KUKA KRL program: MyProgram_062().src

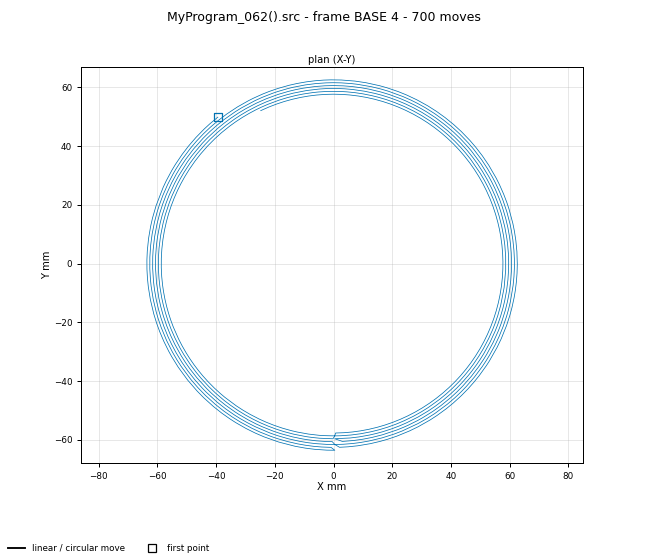
[picture p0: tool path of MyProgram_062().src in frame BASE 4, 700 of 700 moves have a stored position in this frame; points joined in program order, loops and branches not executed]
&ACCESS RVP
&REL 1
&PARAM TEMPLATE = C:\KRC\Roboter\Template\vorgabe
&PARAM EDITMASK = *
DEF MyProgram_062()
; ---- Setting reference (Base) ----
$BASE = BASE_DATA[4]

; --------------------------
; ---- Setting tool (TCP) ----
$TOOL = TOOL_DATA[3]
; --------------------------

$VEL.CP = VEL_APROX_PRINT
Startdeposition()
$VEL.CP = VEL_PRINT
LIN {X -39.4087,Y 49.8917,Z 72,A 123.1029,B 24.8681,C -2.6505,E1 24.8985,E2 -39.1381} C_DIS
LIN {X -42.1841,Y 47.5689,Z 72,A 125.8881,B 24.8698,C -2.6337,E1 24.8927,E2 -41.8942} C_DIS
LIN {X -44.0443,Y 45.8513,Z 72,A 128.1731,B 24.8703,C -2.6285,E1 24.888,E2 -44.1761} C_DIS
LIN {X -46.8498,Y 42.9805,Z 72,A 132.3088,B 24.8701,C -2.63,E1 24.88,E2 -48.3334} C_DIS
LIN {X -49.4029,Y 40.0198,Z 72,A 135.1224,B 24.8724,C -2.6071,E1 24.8751,E2 -51.1051} C_DIS
LIN {X -51.5627,Y 37.1965,Z 72,A 138.8579,B 24.8722,C -2.609,E1 24.8688,E2 -54.8631} C_DIS
LIN {X -53.8773,Y 33.7561,Z 72,A 142.4511,B 24.8735,C -2.5959,E1 24.8633,E2 -58.443} C_DIS
LIN {X -55.0548,Y 31.7997,Z 72,A 145.6129,B 24.8719,C -2.6117,E1 24.8589,E2 -61.6591} C_DIS
LIN {X -56.9529,Y 28.2593,Z 72,A 147.7032,B 24.8759,C -2.5714,E1 24.8563,E2 -63.6644} C_DIS
LIN {X -58.0502,Y 25.9311,Z 72,A 150.8815,B 24.8749,C -2.5811,E1 24.8526,E2 -66.8831} C_DIS
LIN {X -60.4404,Y 19.7284,Z 72,A 157.1125,B 24.8762,C -2.5675,E1 24.8466,E2 -73.1169} C_DIS
LIN {X -61.6489,Y 15.546,Z 72,A 160.584,B 24.8783,C -2.5466,E1 24.8441,E2 -76.5586} C_DIS
LIN {X -62.288,Y 12.7452,Z 72,A 163.2576,B 24.8789,C -2.5401,E1 24.8426,E2 -79.2325} C_DIS
LIN {X -62.9957,Y 8.5937,Z 72,A 167.1763,B 24.8798,C -2.5305,E1 24.8409,E2 -83.1516} C_DIS
LIN {X -63.432,Y 4.3135,Z 72,A 170.8648,B 24.8813,C -2.5146,E1 24.84,E2 -86.8243} C_DIS
LIN {X -63.5665,Y 1.2399,Z 72,A 173.7515,B 24.8819,C -2.508,E1 24.8398,E2 -89.7126} C_DIS
LIN {X -63.5492,Y -1.9301,Z 72,A 176.4044,B 24.8831,C -2.4951,E1 24.8399,E2 -92.3506} C_DIS
LIN {X -63.3815,Y -5.0015,Z 72,A 179.323,B 24.8837,C -2.4892,E1 24.8405,E2 -95.2727} C_DIS
LIN {X -63.0712,Y -8.0176,Z 72,A -178.3475,B 24.8852,C -2.473,E1 24.8412,E2 -97.5774} C_DIS
LIN {X -62.3757,Y -12.3121,Z 72,A -173.4784,B 24.8846,C -2.4792,E1 24.8435,E2 -102.4902} C_DIS
LIN {X -61.1949,Y -17.2459,Z 72,A -169.5379,B 24.887,C -2.4532,E1 24.8462,E2 -106.3916} C_DIS
LIN {X -60.2158,Y -20.4018,Z 72,A -166.3226,B 24.8874,C -2.4491,E1 24.849,E2 -109.6154} C_DIS
LIN {X -59.1943,Y -23.1991,Z 72,A -163.5449,B 24.888,C -2.4432,E1 24.8518,E2 -112.3946} C_DIS
LIN {X -57.8193,Y -26.4415,Z 72,A -160.1766,B 24.8884,C -2.4381,E1 24.8556,E2 -115.7694} C_DIS
LIN {X -56.1547,Y -29.8148,Z 72,A -157.088,B 24.8898,C -2.423,E1 24.8595,E2 -118.8383} C_DIS
LIN {X -55.0992,Y -31.7223,Z 72,A -154.4354,B 24.889,C -2.4315,E1 24.8633,E2 -121.5251} C_DIS
LIN {X -52.8977,Y -35.2725,Z 72,A -150.6395,B 24.8899,C -2.4226,E1 24.8691,E2 -125.3188} C_DIS
LIN {X -49.6828,Y -39.6726,Z 72,A -146.3621,B 24.8921,C -2.3981,E1 24.8762,E2 -129.5581} C_DIS
LIN {X -46.4542,Y -43.4082,Z 72,A -142.251,B 24.8936,C -2.3813,E1 24.8838,E2 -133.6478} C_DIS
LIN {X -44.2089,Y -45.6927,Z 72,A -138.8187,B 24.8931,C -2.3865,E1 24.8906,E2 -137.1067} C_DIS
LIN {X -40.9164,Y -48.6639,Z 72,A -134.084,B 24.8924,C -2.3942,E1 24.9007,E2 -141.8784} C_DIS
LIN {X -38.0706,Y -50.9204,Z 72,A -132.3527,B 24.8958,C -2.3564,E1 24.9044,E2 -143.5259} C_DIS
LIN {X -35.4553,Y -52.775,Z 72,A -129.2005,B 24.8958,C -2.3571,E1 24.9116,E2 -146.6906} C_DIS
LIN {X -33.3423,Y -54.135,Z 72,A -126.1545,B 24.8946,C -2.3702,E1 24.9189,E2 -149.7773} C_DIS
LIN {X -29.7959,Y -56.1647,Z 72,A -122.7593,B 24.8956,C -2.3592,E1 24.9271,E2 -153.156} C_DIS
LIN {X -26.6688,Y -57.7141,Z 72,A -119.8023,B 24.8962,C -2.3515,E1 24.9346,E2 -156.1024} C_DIS
LIN {X -23.6355,Y -59.0214,Z 72,A -116.2682,B 24.8954,C -2.3606,E1 24.9438,E2 -159.6661} C_DIS
LIN {X -18.6731,Y -60.7748,Z 72,A -111.3431,B 24.8954,C -2.3609,E1 24.9568,E2 -164.6009} C_DIS
LIN {X -13.1378,Y -62.2066,Z 72,A -106.4459,B 24.8961,C -2.3526,E1 24.9701,E2 -169.4849} C_DIS
LIN {X -9.5784,Y -62.853,Z 72,A -103.68,B 24.8972,C -2.3406,E1 24.9777,E2 -172.2249} C_DIS
LIN {X -6.4154,Y -63.2537,Z 72,A -100.3205,B 24.8963,C -2.3511,E1 24.9871,E2 -175.6117} C_DIS
LIN {X -2.2636,Y -63.5382,Z 72,A -97.0525,B 24.8972,C -2.3404,E1 24.9961,E2 -178.855} C_DIS
LIN {X 0.4542,Y -63.5727,Z 72,A -95.6125,B 24.8992,C -2.3181,E1 25,E2 -180.2423} C_DIS
Enddeposition()
LIN {X 0.4542,Y -63.5727,Z 72,A -95.6125,B 24.8992,C -2.3181,E1 25,E2 -180.2423} C_DIS
Startdeposition()
$VEL.CP = VEL_PRINT
LIN {X -0.8607,Y -62.5943,Z 72,A -97.3315,B 24.8987,C -2.3237,E1 24.9952,E2 -178.5364} C_DIS
LIN {X -4.0751,Y -62.4673,Z 72,A -99.6734,B 24.8976,C -2.3366,E1 24.9888,E2 -176.2246} C_DIS
LIN {X -6.8501,Y -62.2243,Z 72,A -102.6308,B 24.8983,C -2.328,E1 24.9805,E2 -173.2451} C_DIS
LIN {X -9.5335,Y -61.8698,Z 72,A -104.7295,B 24.8975,C -2.3367,E1 24.9747,E2 -171.1653} C_DIS
LIN {X -12.3094,Y -61.3778,Z 72,A -107.5509,B 24.8979,C -2.3325,E1 24.967,E2 -168.3309} C_DIS
LIN {X -15.6367,Y -60.6156,Z 72,A -111.5838,B 24.8994,C -2.3151,E1 24.9559,E2 -164.251} C_DIS
LIN {X -19.0487,Y -59.6309,Z 72,A -113.7979,B 24.8973,C -2.339,E1 24.9502,E2 -162.0898} C_DIS
LIN {X -21.296,Y -58.8665,Z 72,A -116.4905,B 24.8981,C -2.33,E1 24.943,E2 -159.3706} C_DIS
LIN {X -25.0912,Y -57.3515,Z 72,A -119.7302,B 24.8969,C -2.3441,E1 24.9347,E2 -156.1571} C_DIS
LIN {X -27.7207,Y -56.1277,Z 72,A -122.7428,B 24.8973,C -2.3399,E1 24.9271,E2 -153.1266} C_DIS
LIN {X -31.5587,Y -54.0624,Z 72,A -126.63,B 24.8966,C -2.3473,E1 24.9176,E2 -149.2459} C_DIS
LIN {X -34.5626,Y -52.1938,Z 72,A -130.121,B 24.8966,C -2.3471,E1 24.9094,E2 -145.7432} C_DIS
LIN {X -37.3656,Y -50.2258,Z 72,A -132.5987,B 24.895,C -2.3655,E1 24.9039,E2 -143.3005} C_DIS
LIN {X -40.2209,Y -47.97,Z 72,A -135.7357,B 24.8941,C -2.3753,E1 24.897,E2 -140.1753} C_DIS
LIN {X -43.5614,Y -44.9577,Z 72,A -140.7015,B 24.8949,C -2.3667,E1 24.8867,E2 -135.1691} C_DIS
LIN {X -46.1783,Y -42.265,Z 72,A -144.3865,B 24.8947,C -2.3694,E1 24.8797,E2 -131.4742} C_DIS
LIN {X -48.6608,Y -39.3813,Z 72,A -147.8735,B 24.8939,C -2.3773,E1 24.8735,E2 -127.99} C_DIS
LIN {X -51.8571,Y -35.0657,Z 72,A -152.0596,B 24.8916,C -2.4032,E1 24.8667,E2 -123.8453} C_DIS
LIN {X -53.29,Y -32.8469,Z 72,A -155.0033,B 24.892,C -2.3994,E1 24.8623,E2 -120.8775} C_DIS
LIN {X -54.8561,Y -30.1609,Z 72,A -157.6334,B 24.8909,C -2.4109,E1 24.8587,E2 -118.2612} C_DIS
LIN {X -56.8657,Y -26.173,Z 72,A -162.0699,B 24.8905,C -2.4157,E1 24.8533,E2 -113.812} C_DIS
LIN {X -58.7065,Y -21.7327,Z 72,A -166.1333,B 24.8888,C -2.4345,E1 24.8492,E2 -109.7708} C_DIS
LIN {X -59.7438,Y -18.6938,Z 72,A -168.837,B 24.8876,C -2.4475,E1 24.8468,E2 -107.0827} C_DIS
LIN {X -60.4062,Y -16.4273,Z 72,A -171.656,B 24.8881,C -2.4418,E1 24.8447,E2 -104.2338} C_DIS
LIN {X -61.4194,Y -12.1032,Z 72,A -176.6445,B 24.8885,C -2.4375,E1 24.8418,E2 -99.2056} C_DIS
LIN {X -62.1183,Y -7.7548,Z 72,A -179.0923,B 24.8847,C -2.4787,E1 24.8409,E2 -96.8416} C_DIS
LIN {X -62.3619,Y -5.4582,Z 72,A 178.1174,B 24.8852,C -2.4729,E1 24.8402,E2 -94.0208} C_DIS
LIN {X -62.5753,Y -1.7646,Z 72,A 174.8946,B 24.884,C -2.4865,E1 24.8398,E2 -90.8112} C_DIS
LIN {X -62.5603,Y 2.2343,Z 72,A 171.399,B 24.8826,C -2.5011,E1 24.84,E2 -87.3293} C_DIS
LIN {X -62.2886,Y 6.236,Z 72,A 167.1517,B 24.8825,C -2.5023,E1 24.8409,E2 -83.0593} C_DIS
LIN {X -61.7859,Y 10.066,Z 72,A 163.8912,B 24.8809,C -2.5184,E1 24.8423,E2 -79.8179} C_DIS
LIN {X -60.9672,Y 14.2046,Z 72,A 160.1823,B 24.8795,C -2.5332,E1 24.8444,E2 -76.1227} C_DIS
LIN {X -60.1472,Y 17.3504,Z 72,A 156.9368,B 24.8791,C -2.5375,E1 24.8468,E2 -72.8686} C_DIS
LIN {X -59.3158,Y 20.0098,Z 72,A 153.7977,B 24.8794,C -2.5347,E1 24.8497,E2 -69.7047} C_DIS
LIN {X -58.1418,Y 23.2013,Z 72,A 151.924,B 24.8763,C -2.5667,E1 24.8515,E2 -67.897} C_DIS
LIN {X -56.5004,Y 26.9533,Z 72,A 148.0079,B 24.8756,C -2.5747,E1 24.8559,E2 -63.9784} C_DIS
LIN {X -54.6874,Y 30.4639,Z 72,A 144.1834,B 24.8749,C -2.5812,E1 24.8609,E2 -60.1493} C_DIS
LIN {X -53.7182,Y 32.1435,Z 72,A 141.2134,B 24.8766,C -2.5643,E1 24.8653,E2 -57.1235} C_DIS
LIN {X -51.5773,Y 35.4769,Z 72,A 138.7753,B 24.8735,C -2.596,E1 24.869,E2 -54.7492} C_DIS
LIN {X -48.7578,Y 39.2617,Z 72,A 134.4087,B 24.8724,C -2.6065,E1 24.8763,E2 -50.3867} C_DIS
LIN {X -46.6518,Y 41.7416,Z 72,A 131.2568,B 24.872,C -2.6107,E1 24.8821,E2 -47.2307} C_DIS
LIN {X -44.2997,Y 44.2313,Z 72,A 128.0719,B 24.8714,C -2.6173,E1 24.8883,E2 -44.0477} C_DIS
LIN {X -41.8688,Y 46.5378,Z 72,A 124.9597,B 24.8708,C -2.6235,E1 24.8947,E2 -40.9376} C_DIS
LIN {X -39.2255,Y 48.7871,Z 72,A 120.9549,B 24.8716,C -2.6146,E1 24.9034,E2 -36.8964} C_DIS
LIN {X -36.3682,Y 50.952,Z 72,A 118.6861,B 24.8691,C -2.6406,E1 24.9084,E2 -34.6817} C_DIS
LIN {X -32.678,Y 53.3942,Z 72,A 114.9959,B 24.8676,C -2.6552,E1 24.917,E2 -31.0146} C_DIS
LIN {X -28.963,Y 55.4965,Z 72,A 110.8588,B 24.8674,C -2.6574,E1 24.9271,E2 -26.8705} C_DIS
LIN {X -27.3313,Y 56.3189,Z 72,A 108.0414,B 24.8694,C -2.6374,E1 24.9343,E2 -23.9983} C_DIS
LIN {X -24.1645,Y 57.7483,Z 72,A 106.0643,B 24.8666,C -2.6658,E1 24.9392,E2 -22.0842} C_DIS
LIN {X -21.7428,Y 58.7028,Z 72,A 102.8612,B 24.8679,C -2.6525,E1 24.9477,E2 -18.8426} C_DIS
LIN {X -18.8913,Y 59.6813,Z 72,A 100.1456,B 24.8675,C -2.6565,E1 24.9549,E2 -16.1318} C_DIS
LIN {X -15.152,Y 60.7387,Z 72,A 97.1477,B 24.866,C -2.6714,E1 24.9629,E2 -13.1648} C_DIS
LIN {X -12.5227,Y 61.3346,Z 72,A 94.1782,B 24.8668,C -2.6632,E1 24.9711,E2 -10.1722} C_DIS
LIN {X -9.2487,Y 61.9136,Z 72,A 91.6862,B 24.8655,C -2.6767,E1 24.9778,E2 -7.7101} C_DIS
LIN {X -6.2608,Y 62.2862,Z 72,A 88.4602,B 24.8663,C -2.6685,E1 24.9869,E2 -4.4623} C_DIS
LIN {X -3.3298,Y 62.5115,Z 72,A 86.2742,B 24.8651,C -2.6801,E1 24.9929,E2 -2.3033} C_DIS
LIN {X -0.8723,Y 62.5942,Z 72,A 83.5094,B 24.8661,C -2.6698,E1 25.0007,E2 0.4862} C_DIS
LIN {X 2.6652,Y 62.543,Z 72,A 79.8513,B 24.867,C -2.6613,E1 25.0109,E2 4.1638} C_DIS
LIN {X 7.2533,Y 62.1784,Z 72,A 76.2896,B 24.8657,C -2.6747,E1 25.0207,E2 7.6913} C_DIS
LIN {X 11.0314,Y 61.6203,Z 72,A 72.8045,B 24.8657,C -2.6738,E1 25.0303,E2 11.1751} C_DIS
LIN {X 15.7256,Y 60.5923,Z 72,A 68.4256,B 24.8659,C -2.672,E1 25.0422,E2 15.5523} C_DIS
LIN {X 18.2437,Y 59.8831,Z 72,A 65.6427,B 24.867,C -2.6617,E1 25.0497,E2 18.3548} C_DIS
LIN {X 22.0662,Y 58.582,Z 72,A 62.4765,B 24.8661,C -2.6703,E1 25.058,E2 21.4942} C_DIS
LIN {X 24.8618,Y 57.4515,Z 72,A 59.4177,B 24.8671,C -2.6607,E1 25.0659,E2 24.5686} C_DIS
LIN {X 28.3993,Y 55.7871,Z 72,A 55.7414,B 24.8677,C -2.6541,E1 25.0751,E2 28.2507} C_DIS
LIN {X 32.0976,Y 53.7455,Z 72,A 51.4504,B 24.8692,C -2.639,E1 25.0856,E2 32.5645} C_DIS
LIN {X 35.0671,Y 51.8561,Z 72,A 48.0357,B 24.8702,C -2.6295,E1 25.0935,E2 35.9904} C_DIS
LIN {X 38.0295,Y 49.7248,Z 72,A 45.0496,B 24.87,C -2.6317,E1 25.1001,E2 38.9602} C_DIS
LIN {X 40.9337,Y 47.3633,Z 72,A 41.7935,B 24.8702,C -2.6292,E1 25.107,E2 42.2097} C_DIS
LIN {X 43.548,Y 44.9706,Z 72,A 39.1123,B 24.8695,C -2.6358,E1 25.1124,E2 44.8642} C_DIS
LIN {X 46.4331,Y 41.9858,Z 72,A 34.8017,B 24.8716,C -2.6155,E1 25.1207,E2 49.204} C_DIS
LIN {X 48.4319,Y 39.6632,Z 72,A 31.482,B 24.8734,C -2.5969,E1 25.1266,E2 52.5526} C_DIS
LIN {X 50.6741,Y 36.7555,Z 72,A 29.5115,B 24.8709,C -2.6219,E1 25.1298,E2 54.4543} C_DIS
LIN {X 52.8826,Y 33.5001,Z 72,A 25.7875,B 24.8721,C -2.6099,E1 25.1356,E2 58.1883} C_DIS
LIN {X 55.4247,Y 29.1005,Z 72,A 21.114,B 24.8734,C -2.597,E1 25.1421,E2 62.868} C_DIS
LIN {X 56.547,Y 26.8553,Z 72,A 18.3488,B 24.8751,C -2.5793,E1 25.1455,E2 65.6603} C_DIS
LIN {X 57.9844,Y 23.5916,Z 72,A 15.3849,B 24.8753,C -2.5774,E1 25.1487,E2 68.6125} C_DIS
LIN {X 59.029,Y 20.8404,Z 72,A 12.6504,B 24.8761,C -2.5686,E1 25.1513,E2 71.3525} C_DIS
LIN {X 59.7725,Y 18.6014,Z 72,A 9.9855,B 24.8779,C -2.5498,E1 25.1536,E2 74.0466} C_DIS
LIN {X 61.0954,Y 13.6431,Z 72,A 5.9822,B 24.8777,C -2.5527,E1 25.1563,E2 78.0199} C_DIS
LIN {X 61.6136,Y 11.0689,Z 72,A 3.7892,B 24.8779,C -2.5506,E1 25.1574,E2 80.2051} C_DIS
LIN {X 62.0954,Y 7.9258,Z 72,A 0.4107,B 24.8798,C -2.53,E1 25.1588,E2 83.6126} C_DIS
LIN {X 62.4671,Y 4.0761,Z 72,A -3.3104,B 24.8813,C -2.5144,E1 25.1596,E2 87.3484} C_DIS
LIN {X 62.6,Y -0.1917,Z 72,A -6.6747,B 24.8813,C -2.5155,E1 25.1598,E2 90.69} C_DIS
LIN {X 62.5161,Y -3.2468,Z 72,A -9.7931,B 24.8828,C -2.4987,E1 25.1594,E2 93.8296} C_DIS
LIN {X 62.2941,Y -6.1801,Z 72,A -12.0861,B 24.8827,C -2.5001,E1 25.1589,E2 96.1057} C_DIS
LIN {X 61.9148,Y -9.2354,Z 72,A -15.0389,B 24.8838,C -2.4878,E1 25.1578,E2 99.0701} C_DIS
LIN {X 61.5276,Y -11.5374,Z 72,A -17.3677,B 24.8849,C -2.4763,E1 25.1566,E2 101.4125} C_DIS
LIN {X 60.7674,Y -15.0373,Z 72,A -20.3845,B 24.8853,C -2.4725,E1 25.1547,E2 104.4206} C_DIS
LIN {X 60.0254,Y -17.7675,Z 72,A -23.0144,B 24.8861,C -2.4635,E1 25.1527,E2 107.0568} C_DIS
LIN {X 58.9462,Y -21.0734,Z 72,A -26.5582,B 24.8878,C -2.4448,E1 25.1495,E2 110.6248} C_DIS
LIN {X 57.1353,Y -25.5792,Z 72,A -30.7757,B 24.8885,C -2.4371,E1 25.1449,E2 114.8374} C_DIS
LIN {X 55.7289,Y -28.5139,Z 72,A -34.274,B 24.8905,C -2.4156,E1 25.1405,E2 118.3678} C_DIS
LIN {X 53.0584,Y -33.22,Z 72,A -38.2032,B 24.8895,C -2.4267,E1 25.135,E2 122.2506} C_DIS
LIN {X 52.1163,Y -34.6802,Z 72,A -40.0053,B 24.8904,C -2.4171,E1 25.1322,E2 124.0665} C_DIS
LIN {X 49.6583,Y -38.116,Z 72,A -43.5616,B 24.8906,C -2.4143,E1 25.1264,E2 127.6122} C_DIS
LIN {X 47.8309,Y -40.3853,Z 72,A -46.5328,B 24.8919,C -2.4,E1 25.1211,E2 130.6036} C_DIS
LIN {X 45.7888,Y -42.6851,Z 72,A -49.5818,B 24.8931,C -2.3873,E1 25.1153,E2 133.669} C_DIS
LIN {X 43.5354,Y -44.9827,Z 72,A -52.2506,B 24.8931,C -2.3869,E1 25.11,E2 136.3275} C_DIS
LIN {X 40.7303,Y -47.5376,Z 72,A -55.8059,B 24.894,C -2.3771,E1 25.1026,E2 139.892} C_DIS
LIN {X 38.3574,Y -49.471,Z 72,A -58.6663,B 24.8946,C -2.3697,E1 25.0963,E2 142.7592} C_DIS
LIN {X 35.23,Y -51.7458,Z 72,A -62.4022,B 24.8957,C -2.3579,E1 25.0877,E2 146.5101} C_DIS
LIN {X 32.8782,Y -53.2717,Z 72,A -64.9739,B 24.8961,C -2.353,E1 25.0816,E2 149.0852} C_DIS
LIN {X 28.8443,Y -55.5589,Z 72,A -69.631,B 24.8976,C -2.3362,E1 25.0701,E2 153.7688} C_DIS
LIN {X 25.8402,Y -57.0179,Z 72,A -71.6799,B 24.8959,C -2.3548,E1 25.0651,E2 155.7682} C_DIS
LIN {X 21.5781,Y -58.7636,Z 72,A -75.5966,B 24.8959,C -2.3559,E1 25.055,E2 159.6735} C_DIS
LIN {X 18.3344,Y -59.855,Z 72,A -79.2874,B 24.8973,C -2.3393,E1 25.0451,E2 163.3968} C_DIS
LIN {X 15.8373,Y -60.5637,Z 72,A -81.3397,B 24.8969,C -2.3442,E1 25.0396,E2 165.4342} C_DIS
LIN {X 12.4936,Y -61.3406,Z 72,A -84.1303,B 24.8964,C -2.3493,E1 25.032,E2 168.2088} C_DIS
LIN {X 8.3178,Y -62.0451,Z 72,A -88.061,B 24.8968,C -2.3451,E1 25.0212,E2 172.1454} C_DIS
LIN {X 4.9941,Y -62.4004,Z 72,A -91.6246,B 24.8979,C -2.3321,E1 25.0112,E2 175.7375} C_DIS
LIN {X 2.0567,Y -62.5663,Z 72,A -94.284,B 24.8979,C -2.3319,E1 25.0038,E2 178.3967} C_DIS
LIN {X 2.0567,Y -62.5663,Z 72,A -94.284,B 24.8979,C -2.3319,E1 25.0038,E2 178.3967} C_DIS
Enddeposition()
LIN {X 0.4424,Y -61.6194,Z 72,A -94.8099,B 24.8946,C -2.3694,E1 25.0026,E2 178.8334} C_DIS
Startdeposition()
$VEL.CP = VEL_PRINT
LIN {X 3.293,Y -61.5335,Z 72,A -91.6913,B 24.8936,C -2.3808,E1 25.0113,E2 175.6887} C_DIS
LIN {X 6.3281,Y -61.2955,Z 72,A -89.1713,B 24.8941,C -2.3753,E1 25.0183,E2 173.1833} C_DIS
LIN {X 8.8597,Y -60.9812,Z 72,A -85.9133,B 24.8922,C -2.397,E1 25.0274,E2 169.8766} C_DIS
LIN {X 12.0469,Y -60.4326,Z 72,A -83.4386,B 24.8931,C -2.3872,E1 25.0342,E2 167.4279} C_DIS
LIN {X 16.4999,Y -59.3717,Z 72,A -79.4267,B 24.8931,C -2.3859,E1 25.045,E2 163.4253} C_DIS
LIN {X 20.7143,Y -58.0354,Z 72,A -75.3956,B 24.8929,C -2.389,E1 25.0557,E2 159.3945} C_DIS
LIN {X 23.374,Y -57.016,Z 72,A -72.5319,B 24.8921,C -2.3977,E1 25.0631,E2 156.5167} C_DIS
LIN {X 28.7742,Y -54.4908,Z 72,A -67.1581,B 24.8917,C -2.4024,E1 25.0766,E2 151.1458} C_DIS
LIN {X 31.8208,Y -52.7698,Z 72,A -64.1285,B 24.8917,C -2.4029,E1 25.0839,E2 148.1241} C_DIS
LIN {X 34.5048,Y -51.0551,Z 72,A -60.468,B 24.8896,C -2.4254,E1 25.0926,E2 144.4227} C_DIS
LIN {X 38.7763,Y -47.8915,Z 72,A -56.1143,B 24.89,C -2.4215,E1 25.1021,E2 140.094} C_DIS
LIN {X 41.3572,Y -45.6824,Z 72,A -52.9013,B 24.8892,C -2.4299,E1 25.1089,E2 136.8737} C_DIS
LIN {X 43.5322,Y -43.6148,Z 72,A -50.4166,B 24.8892,C -2.4291,E1 25.1139,E2 134.4013} C_DIS
LIN {X 45.2616,Y -41.8163,Z 72,A -47.9192,B 24.8883,C -2.4391,E1 25.1187,E2 131.8911} C_DIS
LIN {X 48.0068,Y -38.6341,Z 72,A -44.0033,B 24.8874,C -2.4493,E1 25.1257,E2 127.969} C_DIS
LIN {X 50.6737,Y -35.0628,Z 72,A -39.8495,B 24.8864,C -2.4607,E1 25.1326,E2 123.8084} C_DIS
LIN {X 52.0159,Y -33.0396,Z 72,A -37.923,B 24.8865,C -2.4588,E1 25.1355,E2 121.896} C_DIS
LIN {X 53.2021,Y -31.0939,Z 72,A -35.2638,B 24.8847,C -2.4782,E1 25.1393,E2 119.2047} C_DIS
LIN {X 55.0274,Y -27.7343,Z 72,A -32.2869,B 24.8851,C -2.4741,E1 25.1432,E2 116.2529} C_DIS
LIN {X 56.3578,Y -24.9191,Z 72,A -28.8028,B 24.8829,C -2.4974,E1 25.1473,E2 112.7329} C_DIS
LIN {X 57.7739,Y -21.4335,Z 72,A -25.1084,B 24.8815,C -2.5129,E1 25.151,E2 109.0223} C_DIS
LIN {X 58.9461,Y -17.9613,Z 72,A -22.3487,B 24.882,C -2.5071,E1 25.1533,E2 106.2919} C_DIS
LIN {X 59.5578,Y -15.8146,Z 72,A -20.3456,B 24.8816,C -2.5118,E1 25.1548,E2 104.2893} C_DIS
LIN {X 60.2468,Y -12.9414,Z 72,A -16.9379,B 24.8792,C -2.5369,E1 25.1569,E2 100.8418} C_DIS
LIN {X 61.1682,Y -7.4614,Z 72,A -12.2619,B 24.8788,C -2.5409,E1 25.1588,E2 96.1841} C_DIS
LIN {X 61.4634,Y -4.418,Z 72,A -9.4833,B 24.8781,C -2.5483,E1 25.1595,E2 93.4045} C_DIS
LIN {X 61.6017,Y -1.5586,Z 72,A -6.4637,B 24.8764,C -2.5657,E1 25.1598,E2 90.3617} C_DIS
LIN {X 61.5989,Y 1.6666,Z 72,A -4.1806,B 24.8772,C -2.5573,E1 25.1597,E2 88.112} C_DIS
LIN {X 61.4573,Y 4.4916,Z 72,A -1.1094,B 24.8754,C -2.5765,E1 25.1592,E2 85.0136} C_DIS
LIN {X 61.0842,Y 8.119,Z 72,A 2.4249,B 24.874,C -2.5907,E1 25.158,E2 81.4668} C_DIS
LIN {X 60.553,Y 11.426,Z 72,A 5.0789,B 24.8742,C -2.5888,E1 25.1567,E2 78.8328} C_DIS
LIN {X 60.1363,Y 13.4477,Z 72,A 7.4108,B 24.8726,C -2.6049,E1 25.1553,E2 76.4764} C_DIS
LIN {X 59.0332,Y 17.6704,Z 72,A 11.1983,B 24.8721,C -2.6103,E1 25.1525,E2 72.6978} C_DIS
LIN {X 57.676,Y 21.6935,Z 72,A 15.2338,B 24.8707,C -2.6239,E1 25.1487,E2 68.6527} C_DIS
LIN {X 56.5416,Y 24.4988,Z 72,A 18.0173,B 24.87,C -2.6311,E1 25.1457,E2 65.8674} C_DIS
LIN {X 55.1024,Y 27.5861,Z 72,A 20.8147,B 24.87,C -2.6308,E1 25.1424,E2 63.0859} C_DIS
LIN {X 54.1468,Y 29.4162,Z 72,A 23.7492,B 24.8671,C -2.6608,E1 25.1384,E2 60.0957} C_DIS
LIN {X 52.4711,Y 32.312,Z 72,A 25.6755,B 24.8691,C -2.64,E1 25.1357,E2 58.2286} C_DIS
LIN {X 50.4861,Y 35.3319,Z 72,A 29.2782,B 24.8677,C -2.6543,E1 25.1301,E2 54.6099} C_DIS
LIN {X 47.7248,Y 38.982,Z 72,A 33.303,B 24.8673,C -2.6588,E1 25.1232,E2 50.5935} C_DIS
LIN {X 45.9258,Y 41.0855,Z 72,A 36.3387,B 24.8656,C -2.6756,E1 25.1176,E2 47.5316} C_DIS
LIN {X 42.9113,Y 44.2251,Z 72,A 39.7296,B 24.8663,C -2.6686,E1 25.111,E2 44.1718} C_DIS
LIN {X 40.2688,Y 46.6447,Z 72,A 43.5083,B 24.8646,C -2.6857,E1 25.1031,E2 40.3679} C_DIS
LIN {X 37.3257,Y 49.0314,Z 72,A 47.7007,B 24.8623,C -2.7077,E1 25.0938,E2 36.1387} C_DIS
LIN {X 34.4428,Y 51.0971,Z 72,A 50.2908,B 24.8634,C -2.6965,E1 25.088,E2 33.584} C_DIS
LIN {X 31.1518,Y 53.1679,Z 72,A 53.8399,B 24.8631,C -2.7003,E1 25.0795,E2 30.037} C_DIS
LIN {X 28.6727,Y 54.5439,Z 72,A 56.4622,B 24.8627,C -2.7035,E1 25.0731,E2 27.4147} C_DIS
LIN {X 26.3301,Y 55.7131,Z 72,A 59.3059,B 24.8615,C -2.7158,E1 25.0659,E2 24.5493} C_DIS
LIN {X 23.6707,Y 56.8941,Z 72,A 61.9784,B 24.8613,C -2.7178,E1 25.059,E2 21.8782} C_DIS
LIN {X 18.6415,Y 58.734,Z 72,A 66.6013,B 24.8617,C -2.7141,E1 25.0469,E2 17.2736} C_DIS
LIN {X 16.1745,Y 59.4609,Z 72,A 69.8633,B 24.8595,C -2.7351,E1 25.038,E2 13.967} C_DIS
LIN {X 12.9038,Y 60.2554,Z 72,A 71.8664,B 24.8619,C -2.7117,E1 25.0327,E2 12.0222} C_DIS
LIN {X 8.0374,Y 61.095,Z 72,A 76.7686,B 24.8611,C -2.7198,E1 25.0191,E2 7.1054} C_DIS
LIN {X 5.9705,Y 61.3315,Z 72,A 78.9371,B 24.8605,C -2.7251,E1 25.013,E2 4.9257} C_DIS
LIN {X 2.6608,Y 61.564,Z 72,A 81.6397,B 24.8614,C -2.7169,E1 25.0056,E2 2.2438} C_DIS
LIN {X -0.0111,Y 61.6214,Z 72,A 84.4185,B 24.8608,C -2.7227,E1 24.9978,E2 -0.5487} C_DIS
LIN {X -2.5835,Y 61.5673,Z 72,A 86.3775,B 24.8618,C -2.7128,E1 24.9924,E2 -2.4844} C_DIS
LIN {X -6.015,Y 61.3271,Z 72,A 90.3145,B 24.8603,C -2.7269,E1 24.9813,E2 -6.4568} C_DIS
LIN {X -9.5739,Y 60.8734,Z 72,A 93.4785,B 24.8609,C -2.7211,E1 24.9726,E2 -9.6096} C_DIS
LIN {X -13.8436,Y 60.0462,Z 72,A 97.0824,B 24.8622,C -2.7087,E1 24.9628,E2 -13.1881} C_DIS
LIN {X -15.5319,Y 59.632,Z 72,A 98.6849,B 24.8624,C -2.7068,E1 24.9585,E2 -14.7885} C_DIS
LIN {X -19.0868,Y 58.5911,Z 72,A 102.0793,B 24.8629,C -2.702,E1 24.9494,E2 -18.1773} C_DIS
LIN {X -20.8304,Y 57.9936,Z 72,A 104.545,B 24.8616,C -2.7151,E1 24.9429,E2 -20.6791} C_DIS
LIN {X -24.2643,Y 56.6433,Z 72,A 107.5496,B 24.8629,C -2.7017,E1 24.9352,E2 -23.6586} C_DIS
LIN {X -26.8,Y 55.4885,Z 72,A 110.4436,B 24.8627,C -2.7038,E1 24.9278,E2 -26.5649} C_DIS
LIN {X -31.3577,Y 53.0462,Z 72,A 114.2983,B 24.8654,C -2.6769,E1 24.9185,E2 -30.3664} C_DIS
LIN {X -33.4403,Y 51.7589,Z 72,A 117.5929,B 24.8638,C -2.6926,E1 24.9107,E2 -33.709} C_DIS
LIN {X -37.2722,Y 49.0717,Z 72,A 121.9127,B 24.8648,C -2.6832,E1 24.9009,E2 -38.0214} C_DIS
LIN {X -39.843,Y 47.0081,Z 72,A 124.4813,B 24.8664,C -2.6669,E1 24.8955,E2 -40.5611} C_DIS
LIN {X -42.17,Y 44.9321,Z 72,A 127.7734,B 24.8664,C -2.6679,E1 24.8886,E2 -43.8687} C_DIS
LIN {X -44.4139,Y 42.7155,Z 72,A 131.1914,B 24.8661,C -2.6702,E1 24.882,E2 -47.3069} C_DIS
LIN {X -47.6724,Y 39.0462,Z 72,A 135.4264,B 24.8679,C -2.6523,E1 24.8743,E2 -51.5186} C_DIS
LIN {X -50.2791,Y 35.6265,Z 72,A 138.6832,B 24.8703,C -2.6278,E1 24.869,E2 -54.7325} C_DIS
LIN {X -51.9739,Y 33.1044,Z 72,A 142.2846,B 24.8697,C -2.6345,E1 24.8634,E2 -58.3681} C_DIS
LIN {X -53.5263,Y 30.5316,Z 72,A 144.9196,B 24.8708,C -2.6236,E1 24.8597,E2 -60.9907} C_DIS
LIN {X -55.1466,Y 27.4967,Z 72,A 148.0249,B 24.8718,C -2.6126,E1 24.8558,E2 -64.0863} C_DIS
LIN {X -56.9819,Y 23.4582,Z 72,A 151.7849,B 24.8737,C -2.5936,E1 24.8516,E2 -67.8216} C_DIS
LIN {X -58.1857,Y 20.2882,Z 72,A 155.2559,B 24.8741,C -2.5899,E1 24.8482,E2 -71.3033} C_DIS
LIN {X -59.1408,Y 17.3073,Z 72,A 158.6312,B 24.8741,C -2.5896,E1 24.8454,E2 -74.6972} C_DIS
LIN {X -60.1167,Y 13.533,Z 72,A 162.1316,B 24.8754,C -2.576,E1 24.8431,E2 -78.1856} C_DIS
LIN {X -60.9482,Y 9.0903,Z 72,A 166.5285,B 24.8764,C -2.5663,E1 24.8411,E2 -82.5855} C_DIS
LIN {X -61.4507,Y 4.5758,Z 72,A 170.3764,B 24.8783,C -2.546,E1 24.8401,E2 -86.408} C_DIS
LIN {X -61.5777,Y 2.3158,Z 72,A 172.8124,B 24.8783,C -2.5455,E1 24.8398,E2 -88.8574} C_DIS
LIN {X -61.6007,Y -1.599,Z 72,A 176.3491,B 24.8796,C -2.5321,E1 24.8399,E2 -92.3834} C_DIS
LIN {X -61.3299,Y -5.9873,Z 72,A -179.9999,B 24.8816,C -2.5112,E1 24.8407,E2 -96.0064} C_DIS
LIN {X -60.9823,Y -8.8504,Z 72,A -176.2101,B 24.8805,C -2.5235,E1 24.8421,E2 -99.8481} C_DIS
LIN {X -60.4282,Y -12.0684,Z 72,A -173.0311,B 24.8811,C -2.5169,E1 24.8439,E2 -103.0301} C_DIS
LIN {X -59.6384,Y -15.5077,Z 72,A -170.646,B 24.8836,C -2.4902,E1 24.8455,E2 -105.3655} C_DIS
LIN {X -58.8223,Y -18.3618,Z 72,A -168.2141,B 24.8849,C -2.4759,E1 24.8474,E2 -107.7773} C_DIS
LIN {X -57.7758,Y -21.4285,Z 72,A -164.593,B 24.8847,C -2.4785,E1 24.8508,E2 -111.4251} C_DIS
LIN {X -56.3649,Y -24.9032,Z 72,A -161.4957,B 24.8863,C -2.4614,E1 24.8541,E2 -114.4986} C_DIS
LIN {X -55.1867,Y -27.4157,Z 72,A -158.408,B 24.8861,C -2.4639,E1 24.8579,E2 -117.609} C_DIS
LIN {X -53.6625,Y -30.2922,Z 72,A -155.7878,B 24.8875,C -2.448,E1 24.8614,E2 -120.2052} C_DIS
LIN {X -51.706,Y -33.5227,Z 72,A -152.0795,B 24.888,C -2.4428,E1 24.8669,E2 -123.9198} C_DIS
LIN {X -49.5583,Y -36.623,Z 72,A -147.8818,B 24.8876,C -2.4476,E1 24.8738,E2 -128.1496} C_DIS
LIN {X -47.2847,Y -39.5144,Z 72,A -145.1933,B 24.8896,C -2.4255,E1 24.8785,E2 -130.7977} C_DIS
LIN {X -44.7547,Y -42.3586,Z 72,A -141.5998,B 24.8902,C -2.4188,E1 24.8852,E2 -134.391} C_DIS
LIN {X -43.3675,Y -43.7775,Z 72,A -139.5495,B 24.8902,C -2.419,E1 24.8893,E2 -136.4506} C_DIS
LIN {X -39.6704,Y -47.1545,Z 72,A -134.629,B 24.8905,C -2.4153,E1 24.8996,E2 -141.3817} C_DIS
LIN {X -36.6602,Y -49.5308,Z 72,A -131.2398,B 24.8914,C -2.4056,E1 24.9071,E2 -144.7599} C_DIS
LIN {X -33.609,Y -51.6501,Z 72,A -128.2464,B 24.8927,C -2.3908,E1 24.914,E2 -147.7281} C_DIS
LIN {X -31.8463,Y -52.7546,Z 72,A -126.0736,B 24.8926,C -2.3928,E1 24.9192,E2 -149.9124} C_DIS
LIN {X -29.2655,Y -54.2287,Z 72,A -123.0014,B 24.8923,C -2.3955,E1 24.9268,E2 -152.9999} C_DIS
LIN {X -26.6277,Y -55.5713,Z 72,A -120.2987,B 24.8927,C -2.3912,E1 24.9335,E2 -155.6994} C_DIS
LIN {X -21.7331,Y -57.6618,Z 72,A -115.6451,B 24.8937,C -2.3802,E1 24.9455,E2 -160.337} C_DIS
LIN {X -19.1426,Y -58.5729,Z 72,A -112.5287,B 24.8928,C -2.39,E1 24.9539,E2 -163.4828} C_DIS
LIN {X -15.4327,Y -59.6577,Z 72,A -109.8105,B 24.8947,C -2.3692,E1 24.961,E2 -166.1556} C_DIS
LIN {X -11.4757,Y -60.5436,Z 72,A -105.7407,B 24.8943,C -2.3739,E1 24.9722,E2 -170.2416} C_DIS
LIN {X -8.8672,Y -60.9803,Z 72,A -103.252,B 24.8943,C -2.3739,E1 24.9791,E2 -172.7324} C_DIS
LIN {X -6.1503,Y -61.3135,Z 72,A -100.5068,B 24.8939,C -2.378,E1 24.9867,E2 -175.489} C_DIS
LIN {X -2.1776,Y -61.583,Z 72,A -96.959,B 24.8942,C -2.3748,E1 24.9966,E2 -179.0302} C_DIS
LIN {X 0.4424,Y -61.6194,Z 72,A -94.8089,B 24.8947,C -2.369,E1 25.0026,E2 -181.1666} C_DIS
Enddeposition()
LIN {X 0.4424,Y -61.6194,Z 72,A -94.8089,B 24.8947,C -2.369,E1 25.0026,E2 -181.1666} C_DIS
Startdeposition()
$VEL.CP = VEL_PRINT
LIN {X -0.4328,Y -60.6414,Z 72,A -96.3852,B 24.8947,C -2.3695,E1 24.9982,E2 -179.5916} C_DIS
LIN {X -2.7331,Y -60.5813,Z 72,A -98.9926,B 24.8955,C -2.3601,E1 24.9908,E2 -176.9614} C_DIS
LIN {X -5.8894,Y -60.3562,Z 72,A -101.8982,B 24.8953,C -2.362,E1 24.9827,E2 -174.0588} C_DIS
LIN {X -9.0908,Y -59.9579,Z 72,A -104.6176,B 24.8947,C -2.3694,E1 24.9753,E2 -171.355} C_DIS
LIN {X -10.6356,Y -59.703,Z 72,A -107.2508,B 24.8967,C -2.3462,E1 24.9679,E2 -168.664} C_DIS
LIN {X -13.9347,Y -59.0203,Z 72,A -109.4776,B 24.8949,C -2.3672,E1 24.9619,E2 -166.4842} C_DIS
LIN {X -18.0565,Y -57.8924,Z 72,A -113.556,B 24.8947,C -2.3689,E1 24.951,E2 -162.4035} C_DIS
LIN {X -20.6285,Y -57.0268,Z 72,A -116.1965,B 24.8947,C -2.3695,E1 24.944,E2 -159.7592} C_DIS
LIN {X -24.3677,Y -55.532,Z 72,A -120.0469,B 24.8944,C -2.3724,E1 24.9341,E2 -155.907} C_DIS
LIN {X -26.2762,Y -54.6546,Z 72,A -122.1833,B 24.8944,C -2.3717,E1 24.9287,E2 -153.7635} C_DIS
LIN {X -28.9999,Y -53.2595,Z 72,A -124.9843,B 24.894,C -2.3772,E1 24.9218,E2 -150.9677} C_DIS
LIN {X -32.1384,Y -51.4265,Z 72,A -127.8567,B 24.8925,C -2.393,E1 24.9149,E2 -148.1243} C_DIS
LIN {X -33.5087,Y -50.5446,Z 72,A -130.5736,B 24.8944,C -2.3727,E1 24.9085,E2 -145.3501} C_DIS
LIN {X -36.7046,Y -48.2743,Z 72,A -133.427,B 24.8923,C -2.3952,E1 24.9022,E2 -142.5402} C_DIS
LIN {X -38.9375,Y -46.4918,Z 72,A -137.221,B 24.8937,C -2.3795,E1 24.8939,E2 -138.6943} C_DIS
LIN {X -41.5169,Y -44.203,Z 72,A -139.2805,B 24.8911,C -2.4084,E1 24.8898,E2 -136.6954} C_DIS
LIN {X -43.095,Y -42.666,Z 72,A -141.6989,B 24.8913,C -2.4064,E1 24.885,E2 -134.262} C_DIS
LIN {X -46.5456,Y -38.8727,Z 72,A -147.5882,B 24.8921,C -2.398,E1 24.8741,E2 -128.3261} C_DIS
LIN {X -48.8597,Y -35.9208,Z 72,A -150.1623,B 24.8897,C -2.4242,E1 24.8699,E2 -125.802} C_DIS
LIN {X -50.4287,Y -33.6833,Z 72,A -152.5404,B 24.8888,C -2.4343,E1 24.8661,E2 -123.4363} C_DIS
LIN {X -51.8872,Y -31.3894,Z 72,A -155.5178,B 24.8888,C -2.4334,E1 24.8617,E2 -120.4417} C_DIS
LIN {X -54.1033,Y -27.3928,Z 72,A -159.8534,B 24.8878,C -2.4447,E1 24.856,E2 -116.11} C_DIS
LIN {X -55.4885,Y -24.4646,Z 72,A -162.8288,B 24.8869,C -2.4548,E1 24.8526,E2 -113.1424} C_DIS
LIN {X -56.845,Y -21.1242,Z 72,A -166.4192,B 24.8863,C -2.4612,E1 24.8489,E2 -109.5472} C_DIS
LIN {X -58.0089,Y -17.68,Z 72,A -169.6731,B 24.8851,C -2.4745,E1 24.8462,E2 -106.3066} C_DIS
LIN {X -58.8306,Y -14.7153,Z 72,A -173.0985,B 24.8851,C -2.4741,E1 24.8438,E2 -102.8602} C_DIS
LIN {X -59.4918,Y -11.7621,Z 72,A -175.9769,B 24.8843,C -2.4825,E1 24.8422,E2 -99.9848} C_DIS
LIN {X -60.2856,Y -6.5758,Z 72,A 179.848,B 24.8816,C -2.5116,E1 24.8406,E2 -95.8543} C_DIS
LIN {X -60.6178,Y -1.746,Z 72,A 175.3432,B 24.8801,C -2.5271,E1 24.8398,E2 -91.3596} C_DIS
LIN {X -60.5848,Y 2.6542,Z 72,A 170.7876,B 24.8795,C -2.5333,E1 24.84,E2 -86.7912} C_DIS
LIN {X -60.2966,Y 6.4718,Z 72,A 166.7466,B 24.8791,C -2.5373,E1 24.8411,E2 -82.7356} C_DIS
LIN {X -59.954,Y 9.1161,Z 72,A 164.1807,B 24.8785,C -2.5444,E1 24.8421,E2 -80.1714} C_DIS
LIN {X -59.0666,Y 13.7369,Z 72,A 160.2118,B 24.8763,C -2.5667,E1 24.8444,E2 -76.2323} C_DIS
LIN {X -58.3667,Y 16.4588,Z 72,A 157.079,B 24.8763,C -2.5666,E1 24.8467,E2 -73.081} C_DIS
LIN {X -57.0484,Y 20.5684,Z 72,A 153.0859,B 24.875,C -2.5805,E1 24.8502,E2 -69.0985} C_DIS
LIN {X -56.0088,Y 23.251,Z 72,A 150.2692,B 24.8744,C -2.5869,E1 24.8532,E2 -66.2814} C_DIS
LIN {X -54.1509,Y 27.2991,Z 72,A 146.3305,B 24.8727,C -2.604,E1 24.8579,E2 -62.3622} C_DIS
LIN {X -52.7864,Y 29.854,Z 72,A 143.5752,B 24.872,C -2.6115,E1 24.8616,E2 -59.6103} C_DIS
LIN {X -49.763,Y 34.6584,Z 72,A 138.6903,B 24.8696,C -2.6349,E1 24.869,E2 -54.7566} C_DIS
LIN {X -48.27,Y 36.7088,Z 72,A 135.173,B 24.871,C -2.6211,E1 24.8749,E2 -51.1895} C_DIS
LIN {X -44.7539,Y 40.9227,Z 72,A 130.2797,B 24.8692,C -2.6394,E1 24.8838,E2 -46.3177} C_DIS
LIN {X -42.9306,Y 42.8324,Z 72,A 127.6835,B 24.8688,C -2.6435,E1 24.889,E2 -43.7202} C_DIS
LIN {X -39.4157,Y 46.0866,Z 72,A 123.8777,B 24.8664,C -2.6669,E1 24.8968,E2 -39.9551} C_DIS
LIN {X -37.0729,Y 47.9913,Z 72,A 120.3861,B 24.867,C -2.6611,E1 24.9044,E2 -36.4368} C_DIS
LIN {X -35.0605,Y 49.481,Z 72,A 117.5028,B 24.8675,C -2.6563,E1 24.9111,E2 -33.5319} C_DIS
LIN {X -32.3761,Y 51.2779,Z 72,A 115.2898,B 24.8654,C -2.6776,E1 24.9162,E2 -31.3626} C_DIS
LIN {X -29.8954,Y 52.7631,Z 72,A 112.0447,B 24.8659,C -2.6727,E1 24.9241,E2 -28.0962} C_DIS
LIN {X -26.2686,Y 54.6582,Z 72,A 108.2946,B 24.865,C -2.681,E1 24.9334,E2 -24.356} C_DIS
LIN {X -22.8901,Y 56.157,Z 72,A 104.3223,B 24.8654,C -2.6768,E1 24.9437,E2 -20.3646} C_DIS
LIN {X -18.8542,Y 57.6376,Z 72,A 100.0487,B 24.8654,C -2.6775,E1 24.955,E2 -16.0848} C_DIS
LIN {X -15.3634,Y 58.6647,Z 72,A 98.0524,B 24.8622,C -2.7092,E1 24.9602,E2 -14.1606} C_DIS
LIN {X -12.9788,Y 59.2377,Z 72,A 95.3048,B 24.8628,C -2.7027,E1 24.9677,E2 -11.3941} C_DIS
LIN {X -10.3855,Y 59.7472,Z 72,A 92.7515,B 24.8628,C -2.7035,E1 24.9747,E2 -8.84} C_DIS
LIN {X -6.2395,Y 60.3209,Z 72,A 88.4485,B 24.8632,C -2.6988,E1 24.9867,E2 -4.5229} C_DIS
LIN {X -2.9521,Y 60.5712,Z 72,A 86.0454,B 24.8616,C -2.7145,E1 24.9933,E2 -2.1562} C_DIS
LIN {X -0.1188,Y 60.6425,Z 72,A 82.8612,B 24.8626,C -2.7048,E1 25.0022,E2 1.0512} C_DIS
LIN {X 3.3413,Y 60.5507,Z 72,A 79.5244,B 24.8627,C -2.7036,E1 25.0115,E2 4.3898} C_DIS
LIN {X 6.2118,Y 60.324,Z 72,A 77.3279,B 24.8616,C -2.7143,E1 25.0176,E2 6.5598} C_DIS
LIN {X 9.6594,Y 59.868,Z 72,A 73.5503,B 24.8628,C -2.7031,E1 25.0281,E2 10.3605} C_DIS
LIN {X 12.0804,Y 59.4274,Z 72,A 70.6627,B 24.8641,C -2.6903,E1 25.0361,E2 13.275} C_DIS
LIN {X 16.1002,Y 58.4668,Z 72,A 67.5052,B 24.8627,C -2.7038,E1 25.0445,E2 16.3957} C_DIS
LIN {X 18.989,Y 57.5934,Z 72,A 64.2498,B 24.8638,C -2.6929,E1 25.0532,E2 19.6708} C_DIS
LIN {X 22.7628,Y 56.2088,Z 72,A 61.2862,B 24.8623,C -2.7074,E1 25.0608,E2 22.5936} C_DIS
LIN {X 24.9929,Y 55.2528,Z 72,A 58.7379,B 24.8632,C -2.6993,E1 25.0674,E2 25.1549} C_DIS
LIN {X 27.4251,Y 54.087,Z 72,A 55.9233,B 24.8641,C -2.6904,E1 25.0745,E2 27.9833} C_DIS
LIN {X 29.7761,Y 52.83,Z 72,A 53.8507,B 24.8634,C -2.6968,E1 25.0795,E2 30.0345} C_DIS
LIN {X 31.7154,Y 51.6891,Z 72,A 50.9354,B 24.8655,C -2.6762,E1 25.0866,E2 32.9896} C_DIS
LIN {X 34.7349,Y 49.7098,Z 72,A 47.6265,B 24.8658,C -2.673,E1 25.0942,E2 36.295} C_DIS
LIN {X 38.1064,Y 47.1749,Z 72,A 43.8446,B 24.8661,C -2.6704,E1 25.1025,E2 40.0689} C_DIS
LIN {X 40.9781,Y 44.703,Z 72,A 40.4563,B 24.8663,C -2.6678,E1 25.1096,E2 43.45} C_DIS
LIN {X 43.1665,Y 42.5936,Z 72,A 36.7997,B 24.8687,C -2.644,E1 25.1169,E2 47.1475} C_DIS
LIN {X 45.4182,Y 40.1846,Z 72,A 34.5253,B 24.8675,C -2.6563,E1 25.121,E2 49.3826} C_DIS
LIN {X 47.0016,Y 38.3203,Z 72,A 31.617,B 24.8694,C -2.6372,E1 25.1262,E2 52.3226} C_DIS
LIN {X 50.2947,Y 33.882,Z 72,A 26.6297,B 24.8701,C -2.6298,E1 25.1343,E2 57.3032} C_DIS
LIN {X 52.8512,Y 29.7363,Z 72,A 22.4626,B 24.8703,C -2.628,E1 25.1402,E2 61.4532} C_DIS
LIN {X 53.9467,Y 27.7007,Z 72,A 20.372,B 24.8707,C -2.6243,E1 25.1429,E2 63.5416} C_DIS
LIN {X 55.1032,Y 25.3216,Z 72,A 17.4418,B 24.8724,C -2.6072,E1 25.1464,E2 66.4963} C_DIS
LIN {X 56.5551,Y 21.8871,Z 72,A 14.1808,B 24.8728,C -2.6034,E1 25.1498,E2 69.7484} C_DIS
LIN {X 57.532,Y 19.175,Z 72,A 11.5942,B 24.8732,C -2.5987,E1 25.1522,E2 72.3316} C_DIS
LIN {X 58.7031,Y 15.2139,Z 72,A 7.4716,B 24.8749,C -2.5818,E1 25.1553,E2 76.4704} C_DIS
LIN {X 59.372,Y 12.3511,Z 72,A 4.8818,B 24.8752,C -2.5778,E1 25.1569,E2 79.0546} C_DIS
LIN {X 59.9099,Y 9.4007,Z 72,A 2.13,B 24.8759,C -2.5711,E1 25.1581,E2 81.8062} C_DIS
LIN {X 60.294,Y 6.4975,Z 72,A -0.5656,B 24.8766,C -2.5642,E1 25.159,E2 84.5023} C_DIS
LIN {X 60.5324,Y 3.6622,Z 72,A -3.4198,B 24.8778,C -2.5517,E1 25.1596,E2 87.3688} C_DIS
LIN {X 60.6427,Y -0.1862,Z 72,A -6.94,B 24.8786,C -2.5431,E1 25.1598,E2 90.8885} C_DIS
LIN {X 60.5804,Y -2.7526,Z 72,A -9.0574,B 24.8786,C -2.5429,E1 25.1596,E2 92.9939} C_DIS
LIN {X 60.3767,Y -5.6768,Z 72,A -12.2914,B 24.8805,C -2.5229,E1 25.1588,E2 96.2559} C_DIS
LIN {X 60.0163,Y -8.6956,Z 72,A -14.7658,B 24.8805,C -2.5234,E1 25.1579,E2 98.7146} C_DIS
LIN {X 59.6885,Y -10.7166,Z 72,A -16.555,B 24.8807,C -2.5208,E1 25.1571,E2 100.4993} C_DIS
LIN {X 59.2173,Y -13.0728,Z 72,A -19.1282,B 24.8821,C -2.5063,E1 25.1556,E2 103.0918} C_DIS
LIN {X 58.4922,Y -16.0064,Z 72,A -22.5539,B 24.8842,C -2.4838,E1 25.1531,E2 106.551} C_DIS
LIN {X 57.117,Y -20.3764,Z 72,A -26.1205,B 24.8837,C -2.4888,E1 25.15,E2 110.0856} C_DIS
LIN {X 56.1793,Y -22.8352,Z 72,A -29.0676,B 24.8855,C -2.4702,E1 25.1469,E2 113.0603} C_DIS
LIN {X 54.3763,Y -26.8473,Z 72,A -33.2071,B 24.8866,C -2.4583,E1 25.142,E2 117.2056} C_DIS
LIN {X 52.1936,Y -30.877,Z 72,A -36.8742,B 24.8863,C -2.4618,E1 25.137,E2 120.8455} C_DIS
LIN {X 51.1298,Y -32.6088,Z 72,A -39.2456,B 24.8877,C -2.4456,E1 25.1335,E2 123.2431} C_DIS
LIN {X 49.3956,Y -35.1801,Z 72,A -42.4164,B 24.889,C -2.432,E1 25.1283,E2 126.4307} C_DIS
LIN {X 46.9372,Y -38.3995,Z 72,A -46.0773,B 24.8896,C -2.4259,E1 25.122,E2 130.0888} C_DIS
LIN {X 43.9782,Y -41.756,Z 72,A -49.922,B 24.8896,C -2.4244,E1 25.1148,E2 133.9202} C_DIS
LIN {X 42.0357,Y -43.71,Z 72,A -52.5258,B 24.8903,C -2.4182,E1 25.1096,E2 136.5277} C_DIS
LIN {X 39.9964,Y -45.5837,Z 72,A -55.5999,B 24.8918,C -2.4016,E1 25.1031,E2 139.6287} C_DIS
LIN {X 36.4998,Y -48.4286,Z 72,A -60.2143,B 24.8933,C -2.3844,E1 25.0929,E2 144.2667} C_DIS
LIN {X 33.7797,Y -50.3643,Z 72,A -62.5534,B 24.8922,C -2.3968,E1 25.0876,E2 146.5686} C_DIS
LIN {X 30.3238,Y -52.517,Z 72,A -66.1914,B 24.8924,C -2.3946,E1 25.0789,E2 150.2006} C_DIS
LIN {X 28.6173,Y -53.4668,Z 72,A -69.1821,B 24.895,C -2.3656,E1 25.0714,E2 153.2514} C_DIS
LIN {X 25.356,Y -55.0873,Z 72,A -71.2497,B 24.8927,C -2.3911,E1 25.0664,E2 155.2532} C_DIS
LIN {X 23.9446,Y -55.7157,Z 72,A -72.9897,B 24.8935,C -2.3826,E1 25.0619,E2 157.0092} C_DIS
LIN {X 21.7133,Y -56.6223,Z 72,A -75.3765,B 24.894,C -2.377,E1 25.0556,E2 159.4039} C_DIS
LIN {X 16.6781,Y -58.3046,Z 72,A -80.2431,B 24.8942,C -2.3743,E1 25.0427,E2 164.2677} C_DIS
LIN {X 13.0994,Y -59.2108,Z 72,A -83.6156,B 24.8942,C -2.3735,E1 25.0336,E2 167.6373} C_DIS
LIN {X 10.0698,Y -59.801,Z 72,A -86.7973,B 24.895,C -2.3654,E1 25.0248,E2 170.8347} C_DIS
LIN {X 6.8718,Y -60.2524,Z 72,A -89.7757,B 24.895,C -2.365,E1 25.0166,E2 173.8116} C_DIS
LIN {X 3.0336,Y -60.5674,Z 72,A -93.89,B 24.8961,C -2.3533,E1 25.005,E2 177.952} C_DIS
LIN {X 3.0336,Y -60.5674,Z 72,A -93.89,B 24.8961,C -2.3533,E1 25.005,E2 177.952} C_DIS
Enddeposition()
LIN {X 0.4201,Y -59.6513,Z 72,A -94.4602,B 24.891,C -2.4102,E1 25.0038,E2 178.3868} C_DIS
Startdeposition()
$VEL.CP = VEL_PRINT
LIN {X 5.6808,Y -59.3935,Z 72,A -89.9673,B 24.8919,C -2.3999,E1 25.0163,E2 173.9201} C_DIS
LIN {X 8.7603,Y -59.0186,Z 72,A -86.0321,B 24.8898,C -2.4227,E1 25.0273,E2 169.9342} C_DIS
LIN {X 12.1723,Y -58.4098,Z 72,A -83.5271,B 24.8912,C -2.4074,E1 25.034,E2 167.4686} C_DIS
LIN {X 14.5244,Y -57.8697,Z 72,A -80.9125,B 24.8904,C -2.4161,E1 25.0412,E2 164.8369} C_DIS
LIN {X 16.7736,Y -57.2582,Z 72,A -78.9722,B 24.8908,C -2.4119,E1 25.0464,E2 162.9098} C_DIS
LIN {X 19.9919,Y -56.2152,Z 72,A -75.4957,B 24.89,C -2.421,E1 25.0556,E2 159.4186} C_DIS
LIN {X 22.4462,Y -55.2811,Z 72,A -73.0546,B 24.8899,C -2.4226,E1 25.0619,E2 156.9791} C_DIS
LIN {X 24.9023,Y -54.219,Z 72,A -69.6744,B 24.8878,C -2.445,E1 25.0707,E2 153.5543} C_DIS
LIN {X 28.792,Y -52.2584,Z 72,A -65.9324,B 24.8881,C -2.4418,E1 25.0798,E2 149.8304} C_DIS
LIN {X 32.3129,Y -50.157,Z 72,A -62.5842,B 24.8887,C -2.4355,E1 25.0877,E2 146.5076} C_DIS
LIN {X 34.5826,Y -48.6199,Z 72,A -59.3252,B 24.8869,C -2.4553,E1 25.0953,E2 143.213} C_DIS
LIN {X 37.4183,Y -46.473,Z 72,A -56.1152,B 24.8866,C -2.4578,E1 25.1023,E2 140.0091} C_DIS
LIN {X 39.9178,Y -44.3444,Z 72,A -53.1353,B 24.8863,C -2.4608,E1 25.1086,E2 137.0337} C_DIS
LIN {X 42.1042,Y -42.2745,Z 72,A -50.2455,B 24.8857,C -2.4676,E1 25.1144,E2 134.1399} C_DIS
LIN {X 43.8194,Y -40.4937,Z 72,A -47.865,B 24.8852,C -2.4736,E1 25.1189,E2 131.7557} C_DIS
LIN {X 45.8625,Y -38.1637,Z 72,A -45.0042,B 24.8847,C -2.4785,E1 25.1241,E2 128.8963} C_DIS
LIN {X 47.1397,Y -36.575,Z 72,A -42.9215,B 24.8839,C -2.4866,E1 25.1277,E2 126.8042} C_DIS
LIN {X 48.8024,Y -34.3254,Z 72,A -40.7082,B 24.8843,C -2.4825,E1 25.1313,E2 124.6112} C_DIS
LIN {X 50.0613,Y -32.461,Z 72,A -38.114,B 24.8828,C -2.4989,E1 25.1353,E2 121.9913} C_DIS
LIN {X 51.1848,Y -30.66,Z 72,A -35.9406,B 24.8819,C -2.5078,E1 25.1385,E2 119.8078} C_DIS
LIN {X 53.3033,Y -26.8072,Z 72,A -31.9998,B 24.8814,C -2.5133,E1 25.1437,E2 115.8749} C_DIS
LIN {X 55.0655,Y -22.9709,Z 72,A -28.0062,B 24.8804,C -2.5239,E1 25.1482,E2 111.878} C_DIS
LIN {X 55.9798,Y -20.6426,Z 72,A -25.5091,B 24.8795,C -2.5335,E1 25.1507,E2 109.3721} C_DIS
LIN {X 56.9409,Y -17.8202,Z 72,A -22.9374,B 24.8793,C -2.5352,E1 25.1529,E2 106.8109} C_DIS
LIN {X 57.7177,Y -15.1169,Z 72,A -20.3419,B 24.8788,C -2.541,E1 25.1549,E2 104.2165} C_DIS
LIN {X 58.2789,Y -12.7816,Z 72,A -17.57,B 24.877,C -2.5595,E1 25.1566,E2 101.4169} C_DIS
LIN {X 58.964,Y -9.1147,Z 72,A -14.2564,B 24.8766,C -2.5643,E1 25.1582,E2 98.1115} C_DIS
LIN {X 59.4192,Y -5.4038,Z 72,A -10.1145,B 24.8741,C -2.5891,E1 25.1594,E2 93.9355} C_DIS
LIN {X 59.6331,Y -1.9327,Z 72,A -7.5778,B 24.875,C -2.5801,E1 25.1597,E2 91.435} C_DIS
LIN {X 59.6612,Y 0.6171,Z 72,A -4.8267,B 24.8736,C -2.5952,E1 25.1597,E2 88.6647} C_DIS
LIN {X 59.5621,Y 3.4976,Z 72,A -2.0863,B 24.8728,C -2.6032,E1 25.1594,E2 85.9216} C_DIS
LIN {X 59.2819,Y 6.748,Z 72,A 0.7948,B 24.8724,C -2.6069,E1 25.1586,E2 83.0488} C_DIS
LIN {X 59.0477,Y 8.5564,Z 72,A 2.9529,B 24.8709,C -2.6222,E1 25.1577,E2 80.8674} C_DIS
LIN {X 58.3392,Y 12.5059,Z 72,A 6.2883,B 24.8709,C -2.6215,E1 25.156,E2 77.5532} C_DIS
LIN {X 57.1759,Y 17.0516,Z 72,A 11.0739,B 24.869,C -2.6417,E1 25.1525,E2 72.7473} C_DIS
LIN {X 56.2936,Y 19.7704,Z 72,A 13.7361,B 24.8684,C -2.6477,E1 25.1502,E2 70.0859} C_DIS
LIN {X 55.0206,Y 23.0777,Z 72,A 17.293,B 24.867,C -2.6611,E1 25.1465,E2 66.5169} C_DIS
LIN {X 53.8086,Y 25.7774,Z 72,A 19.981,B 24.8666,C -2.6653,E1 25.1433,E2 63.8335} C_DIS
LIN {X 52.4556,Y 28.4297,Z 72,A 22.9842,B 24.8655,C -2.6764,E1 25.1394,E2 60.8198} C_DIS
LIN {X 50.7483,Y 31.377,Z 72,A 25.9998,B 24.8652,C -2.6789,E1 25.1351,E2 57.8138} C_DIS
LIN {X 49.0147,Y 34.0205,Z 72,A 29.4911,B 24.8634,C -2.6972,E1 25.1295,E2 54.2964} C_DIS
LIN {X 47.4219,Y 36.2085,Z 72,A 31.882,B 24.8632,C -2.6986,E1 25.1255,E2 51.9137} C_DIS
LIN {X 45.5457,Y 38.5417,Z 72,A 34.3368,B 24.8636,C -2.6954,E1 25.1212,E2 49.4777} C_DIS
LIN {X 43.2798,Y 41.0703,Z 72,A 37.7964,B 24.8624,C -2.7071,E1 25.1147,E2 46.0056} C_DIS
LIN {X 41.1644,Y 43.1902,Z 72,A 40.6286,B 24.8619,C -2.7121,E1 25.109,E2 43.1736} C_DIS
LIN {X 38.9584,Y 45.1906,Z 72,A 43.9894,B 24.8601,C -2.7291,E1 25.1019,E2 39.7858} C_DIS
LIN {X 35.815,Y 47.7192,Z 72,A 47.4932,B 24.8603,C -2.7275,E1 25.0942,E2 36.2985} C_DIS
LIN {X 33.2058,Y 49.5711,Z 72,A 50.5935,B 24.8597,C -2.7331,E1 25.087,E2 33.1956} C_DIS
LIN {X 30.1285,Y 51.4991,Z 72,A 53.7056,B 24.86,C -2.7299,E1 25.0797,E2 30.1008} C_DIS
LIN {X 27.3493,Y 53.0264,Z 72,A 57.0481,B 24.8589,C -2.7405,E1 25.0714,E2 26.7427} C_DIS
LIN {X 24.5107,Y 54.3968,Z 72,A 60.1272,B 24.8585,C -2.7451,E1 25.0636,E2 23.6605} C_DIS
LIN {X 21.8497,Y 55.5196,Z 72,A 62.5326,B 24.859,C -2.7398,E1 25.0574,E2 21.2731} C_DIS
LIN {X 19.0368,Y 56.5459,Z 72,A 65.593,B 24.8583,C -2.7463,E1 25.0493,E2 18.2035} C_DIS
LIN {X 16.3488,Y 57.3808,Z 72,A 68.2515,B 24.8583,C -2.7473,E1 25.0422,E2 15.5473} C_DIS
LIN {X 14.041,Y 57.9888,Z 72,A 70.9479,B 24.8572,C -2.7573,E1 25.0349,E2 12.8312} C_DIS
LIN {X 10.5219,Y 58.7293,Z 72,A 75.2309,B 24.8552,C -2.7763,E1 25.023,E2 8.5076} C_DIS
LIN {X 6.4543,Y 59.3145,Z 72,A 77.587,B 24.8586,C -2.7435,E1 25.0167,E2 6.2315} C_DIS
LIN {X 3.8136,Y 59.5426,Z 72,A 80.7214,B 24.8574,C -2.7558,E1 25.0079,E2 3.0692} C_DIS
LIN {X 1.1291,Y 59.6535,Z 72,A 84.1259,B 24.8556,C -2.7727,E1 24.9983,E2 -0.3748} C_DIS
LIN {X -2.5886,Y 59.6082,Z 72,A 86.6509,B 24.858,C -2.75,E1 24.9914,E2 -2.8463} C_DIS
LIN {X -4.8839,Y 59.4642,Z 72,A 89.2427,B 24.8573,C -2.7568,E1 24.9841,E2 -5.4554} C_DIS
LIN {X -9.1543,Y 58.9579,Z 72,A 92.6281,B 24.8591,C -2.7393,E1 24.9748,E2 -8.8017} C_DIS
LIN {X -13.7436,Y 58.0599,Z 72,A 97.49,B 24.8587,C -2.7429,E1 24.9615,E2 -13.6779} C_DIS
LIN {X -16.5291,Y 57.329,Z 72,A 99.9898,B 24.8595,C -2.7349,E1 24.9548,E2 -16.1624} C_DIS
LIN {X -18.9887,Y 56.5621,Z 72,A 102.984,B 24.8588,C -2.7422,E1 24.9468,E2 -19.1794} C_DIS
LIN {X -22.9376,Y 55.0795,Z 72,A 106.8972,B 24.8596,C -2.7341,E1 24.9366,E2 -23.0818} C_DIS
LIN {X -25.7373,Y 53.8279,Z 72,A 110.3042,B 24.8591,C -2.7386,E1 24.928,E2 -26.508} C_DIS
LIN {X -29.2322,Y 52.0129,Z 72,A 113.5989,B 24.8608,C -2.7229,E1 24.92,E2 -29.7747} C_DIS
LIN {X -31.7498,Y 50.5155,Z 72,A 116.3389,B 24.8614,C -2.7164,E1 24.9135,E2 -32.5077} C_DIS
LIN {X -33.5546,Y 49.335,Z 72,A 118.7566,B 24.8612,C -2.719,E1 24.9078,E2 -34.9396} C_DIS
LIN {X -36.5691,Y 47.1441,Z 72,A 122.4865,B 24.8616,C -2.7145,E1 24.8995,E2 -38.6721} C_DIS
LIN {X -39.4534,Y 44.7587,Z 72,A 125.8794,B 24.8628,C -2.7028,E1 24.8923,E2 -42.0504} C_DIS
LIN {X -42.0888,Y 42.2897,Z 72,A 128.8417,B 24.8646,C -2.6854,E1 24.8864,E2 -44.9835} C_DIS
LIN {X -43.9862,Y 40.3119,Z 72,A 132.2966,B 24.8637,C -2.6941,E1 24.8798,E2 -48.4742} C_DIS
LIN {X -46.5725,Y 37.2954,Z 72,A 136.3876,B 24.8642,C -2.6893,E1 24.8725,E2 -52.5728} C_DIS
LIN {X -48.9238,Y 34.1512,Z 72,A 139.2236,B 24.8669,C -2.6623,E1 24.868,E2 -55.358} C_DIS
LIN {X -50.971,Y 31.0127,Z 72,A 143.0628,B 24.8675,C -2.6566,E1 24.8622,E2 -59.2031} C_DIS
LIN {X -52.2984,Y 28.7195,Z 72,A 145.6682,B 24.8681,C -2.6505,E1 24.8587,E2 -61.8075} C_DIS
LIN {X -53.2914,Y 26.8305,Z 72,A 148.2605,B 24.8677,C -2.6543,E1 24.8554,E2 -64.4227} C_DIS
LIN {X -55.035,Y 23.0436,Z 72,A 151.5202,B 24.8702,C -2.6291,E1 24.8517,E2 -67.6403} C_DIS
LIN {X -55.9023,Y 20.8507,Z 72,A 154.6395,B 24.8694,C -2.6375,E1 24.8486,E2 -70.7971} C_DIS
LIN {X -57.2803,Y 16.6973,Z 72,A 158.2509,B 24.8717,C -2.614,E1 24.8457,E2 -74.3732} C_DIS
LIN {X -58.0325,Y 13.8583,Z 72,A 161.0659,B 24.8726,C -2.6052,E1 24.8437,E2 -77.1834} C_DIS
LIN {X -58.9087,Y 9.4723,Z 72,A 165.2663,B 24.8741,C -2.59,E1 24.8416,E2 -81.3724} C_DIS
LIN {X -59.4282,Y 5.3053,Z 72,A 169.4213,B 24.8751,C -2.5794,E1 24.8403,E2 -85.527} C_DIS
LIN {X -59.6226,Y 2.2439,Z 72,A 172.9427,B 24.8751,C -2.5803,E1 24.8398,E2 -89.0717} C_DIS
LIN {X -59.6252,Y -2.1693,Z 72,A 176.8432,B 24.8769,C -2.5609,E1 24.84,E2 -92.9494} C_DIS
LIN {X -59.4391,Y -5.1835,Z 72,A 179.6095,B 24.878,C -2.5495,E1 24.8406,E2 -95.7049} C_DIS
LIN {X -59.1231,Y -8.0217,Z 72,A -176.6006,B 24.877,C -2.5597,E1 24.842,E2 -99.542} C_DIS
LIN {X -58.5275,Y -11.5941,Z 72,A -174.4982,B 24.8804,C -2.5245,E1 24.843,E2 -101.5726} C_DIS
LIN {X -58.0182,Y -13.9184,Z 72,A -171.894,B 24.8804,C -2.5232,E1 24.8446,E2 -104.189} C_DIS
LIN {X -57.3038,Y -16.6162,Z 72,A -169.0638,B 24.881,C -2.5179,E1 24.8467,E2 -107.023} C_DIS
LIN {X -56.3812,Y -19.5193,Z 72,A -166.1923,B 24.8819,C -2.5084,E1 24.8493,E2 -109.8881} C_DIS
LIN {X -55.3618,Y -22.2477,Z 72,A -163.1527,B 24.8822,C -2.5047,E1 24.8524,E2 -112.9361} C_DIS
LIN {X -54.0035,Y -25.3673,Z 72,A -159.6304,B 24.8827,C -2.5003,E1 24.8565,E2 -116.4671} C_DIS
LIN {X -52.257,Y -28.7944,Z 72,A -156.3419,B 24.8843,C -2.4829,E1 24.8607,E2 -119.7316} C_DIS
LIN {X -51.0095,Y -30.9494,Z 72,A -153.9651,B 24.8849,C -2.4765,E1 24.8641,E2 -122.1051} C_DIS
LIN {X -48.7195,Y -34.4422,Z 72,A -150.1074,B 24.8861,C -2.4636,E1 24.8701,E2 -125.9514} C_DIS
LIN {X -46.7392,Y -37.0848,Z 72,A -146.779,B 24.8865,C -2.459,E1 24.8757,E2 -129.2846} C_DIS
LIN {X -45.2104,Y -38.9347,Z 72,A -143.8277,B 24.8859,C -2.4659,E1 24.8812,E2 -132.266} C_DIS
LIN {X -42.4575,Y -41.9189,Z 72,A -140.5179,B 24.8877,C -2.4465,E1 24.8875,E2 -135.5437} C_DIS
LIN {X -40.1053,Y -44.1758,Z 72,A -136.7727,B 24.8872,C -2.452,E1 24.8952,E2 -139.3172} C_DIS
LIN {X -37.2666,Y -46.5953,Z 72,A -133.7617,B 24.8888,C -2.4344,E1 24.9016,E2 -142.2978} C_DIS
LIN {X -35.2481,Y -48.1395,Z 72,A -131.3279,B 24.8892,C -2.4301,E1 24.9071,E2 -144.73} C_DIS
LIN {X -32.5023,Y -50.0354,Z 72,A -128.2233,B 24.8898,C -2.4231,E1 24.9142,E2 -147.8283} C_DIS
LIN {X -30.0269,Y -51.5573,Z 72,A -125.2952,B 24.8899,C -2.4218,E1 24.9213,E2 -150.7623} C_DIS
LIN {X -27.4843,Y -52.9569,Z 72,A -122.3466,B 24.8899,C -2.4214,E1 24.9285,E2 -153.7181} C_DIS
LIN {X -24.9634,Y -54.1908,Z 72,A -119.9662,B 24.8908,C -2.4121,E1 24.9345,E2 -156.0824} C_DIS
LIN {X -22.2279,Y -55.3696,Z 72,A -116.9227,B 24.8908,C -2.4128,E1 24.9424,E2 -159.1346} C_DIS
LIN {X -19.6036,Y -56.3521,Z 72,A -114.1509,B 24.8908,C -2.4122,E1 24.9497,E2 -161.9103} C_DIS
LIN {X -16.9574,Y -57.2039,Z 72,A -111.2726,B 24.8906,C -2.4145,E1 24.9574,E2 -164.7992} C_DIS
LIN {X -13.5679,Y -58.1014,Z 72,A -107.5556,B 24.8901,C -2.42,E1 24.9675,E2 -168.5343} C_DIS
LIN {X -9.3148,Y -58.9331,Z 72,A -104.1569,B 24.8917,C -2.4027,E1 24.9768,E2 -171.8954} C_DIS
LIN {X -7.2248,Y -59.2255,Z 72,A -101.8212,B 24.8911,C -2.4088,E1 24.9833,E2 -174.2473} C_DIS
LIN {X -4.729,Y -59.4766,Z 72,A -99.2409,B 24.8908,C -2.4124,E1 24.9905,E2 -176.8373} C_DIS
LIN {X -0.1795,Y -59.6644,Z 72,A -94.4865,B 24.89,C -2.4213,E1 25.0038,E2 -181.6132} C_DIS
LIN {X -0.1795,Y -59.6644,Z 72,A -94.4865,B 24.89,C -2.4213,E1 25.0038,E2 -181.6132} C_DIS
Enddeposition()
LIN {X 0.4154,Y -58.6803,Z 72,A -95.4263,B 24.8913,C -2.4062,E1 25.0011,E2 -180.6377} C_DIS
Startdeposition()
$VEL.CP = VEL_PRINT
LIN {X -3.3708,Y -58.5891,Z 72,A -99.3499,B 24.8918,C -2.401,E1 24.9901,E2 -176.7011} C_DIS
LIN {X -4.9648,Y -58.4761,Z 72,A -101.576,B 24.893,C -2.3876,E1 24.9838,E2 -174.4421} C_DIS
LIN {X -8.5525,Y -58.0598,Z 72,A -104.7,B 24.8922,C -2.3963,E1 24.9752,E2 -171.3365} C_DIS
LIN {X -12.3739,Y -57.3666,Z 72,A -108.1711,B 24.8915,C -2.4041,E1 24.9657,E2 -167.8802} C_DIS
LIN {X -14.3965,Y -56.893,Z 72,A -110.6662,B 24.8923,C -2.3959,E1 24.9589,E2 -165.3623} C_DIS
LIN {X -17.3464,Y -56.0636,Z 72,A -113.5824,B 24.892,C -2.3994,E1 24.9511,E2 -162.4495} C_DIS
LIN {X -20.2093,Y -55.0965,Z 72,A -116.5034,B 24.8917,C -2.4024,E1 24.9434,E2 -159.53} C_DIS
LIN {X -22.928,Y -54.0218,Z 72,A -119.3426,B 24.8914,C -2.4055,E1 24.9361,E2 -156.6918} C_DIS
LIN {X -25.2587,Y -52.9722,Z 72,A -122.9144,B 24.893,C -2.3881,E1 24.9269,E2 -153.0694} C_DIS
LIN {X -28.4682,Y -51.3187,Z 72,A -125.3291,B 24.8907,C -2.4134,E1 24.9211,E2 -150.7083} C_DIS
LIN {X -30.8305,Y -49.9359,Z 72,A -128.0351,B 24.8904,C -2.4166,E1 24.9147,E2 -148.0016} C_DIS
LIN {X -33.0921,Y -48.4664,Z 72,A -131.0393,B 24.8907,C -2.4139,E1 24.9076,E2 -144.9809} C_DIS
LIN {X -37.0303,Y -45.528,Z 72,A -135.1517,B 24.8887,C -2.4348,E1 24.8986,E2 -140.9035} C_DIS
LIN {X -38.557,Y -44.2424,Z 72,A -137.5473,B 24.8892,C -2.4303,E1 24.8935,E2 -138.4879} C_DIS
LIN {X -40.6613,Y -42.3166,Z 72,A -140.3599,B 24.8887,C -2.4354,E1 24.8877,E2 -135.6759} C_DIS
LIN {X -42.738,Y -40.218,Z 72,A -143.2646,B 24.8882,C -2.4411,E1 24.8821,E2 -132.7722} C_DIS
LIN {X -44.5622,Y -38.1872,Z 72,A -145.7388,B 24.8873,C -2.4504,E1 24.8776,E2 -130.3092} C_DIS
LIN {X -46.0675,Y -36.3567,Z 72,A -148.2297,B 24.8871,C -2.4526,E1 24.8732,E2 -127.812} C_DIS
LIN {X -47.4659,Y -34.5116,Z 72,A -150.7842,B 24.8871,C -2.4529,E1 24.869,E2 -125.2458} C_DIS
LIN {X -49.0107,Y -32.2797,Z 72,A -152.8984,B 24.8856,C -2.4689,E1 24.8657,E2 -123.1592} C_DIS
LIN {X -50.1802,Y -30.4299,Z 72,A -155.3167,B 24.8856,C -2.4695,E1 24.8621,E2 -120.7299} C_DIS
LIN {X -51.5749,Y -28.0009,Z 72,A -158.0293,B 24.8848,C -2.4771,E1 24.8584,E2 -118.0213} C_DIS
LIN {X -52.7845,Y -25.6489,Z 72,A -160.6447,B 24.8842,C -2.4836,E1 24.8552,E2 -115.4072} C_DIS
LIN {X -54.581,Y -21.5628,Z 72,A -164.896,B 24.8829,C -2.4977,E1 24.8505,E2 -111.1661} C_DIS
LIN {X -55.4426,Y -19.2397,Z 72,A -167.345,B 24.8823,C -2.5042,E1 24.8482,E2 -108.7188} C_DIS
LIN {X -56.1913,Y -16.9287,Z 72,A -169.7296,B 24.8817,C -2.5109,E1 24.8462,E2 -106.3367} C_DIS
LIN {X -56.8451,Y -14.5828,Z 72,A -172.1202,B 24.881,C -2.5178,E1 24.8445,E2 -103.9486} C_DIS
LIN {X -57.4322,Y -12.0676,Z 72,A -174.4562,B 24.88,C -2.5286,E1 24.843,E2 -101.6247} C_DIS
LIN {X -57.9061,Y -9.5352,Z 72,A -177.0214,B 24.8793,C -2.5355,E1 24.8418,E2 -99.0607} C_DIS
LIN {X -58.2244,Y -7.3475,Z 72,A -179.5441,B 24.8793,C -2.536,E1 24.8408,E2 -96.5241} C_DIS
LIN {X -58.5193,Y -4.424,Z 72,A 177.554,B 24.8785,C -2.5444,E1 24.8401,E2 -93.6249} C_DIS
LIN {X -58.6695,Y -1.3901,Z 72,A 174.3644,B 24.8779,C -2.55,E1 24.8398,E2 -90.4294} C_DIS
LIN {X -58.6572,Y 1.8322,Z 72,A 171.3991,B 24.8767,C -2.5629,E1 24.8399,E2 -87.4773} C_DIS
LIN {X -58.4778,Y 4.9437,Z 72,A 168.3585,B 24.8758,C -2.5726,E1 24.8405,E2 -84.4414} C_DIS
LIN {X -58.1091,Y 8.2072,Z 72,A 165.1227,B 24.8748,C -2.5822,E1 24.8416,E2 -81.2093} C_DIS
LIN {X -57.5932,Y 11.2729,Z 72,A 162.0586,B 24.8739,C -2.5912,E1 24.8432,E2 -78.1486} C_DIS
LIN {X -56.9392,Y 14.2117,Z 72,A 159.2112,B 24.8729,C -2.6019,E1 24.845,E2 -75.3101} C_DIS
LIN {X -56.2115,Y 16.8614,Z 72,A 156.4028,B 24.8723,C -2.6081,E1 24.8471,E2 -72.5002} C_DIS
LIN {X -55.3716,Y 19.4426,Z 72,A 153.5742,B 24.8718,C -2.6132,E1 24.8497,E2 -69.6677} C_DIS
LIN {X -54.2604,Y 22.3572,Z 72,A 150.7277,B 24.8706,C -2.6257,E1 24.8526,E2 -66.8352} C_DIS
LIN {X -53.1657,Y 24.8484,Z 72,A 147.9945,B 24.8699,C -2.6323,E1 24.8558,E2 -64.1027} C_DIS
LIN {X -52.0399,Y 27.1269,Z 72,A 145.6525,B 24.869,C -2.6418,E1 24.8587,E2 -61.7709} C_DIS
LIN {X -50.7191,Y 29.5245,Z 72,A 142.7883,B 24.8685,C -2.6461,E1 24.8626,E2 -58.9021} C_DIS
LIN {X -49.132,Y 32.0957,Z 72,A 139.302,B 24.8686,C -2.6452,E1 24.8679,E2 -55.3958} C_DIS
LIN {X -47.1901,Y 34.8883,Z 72,A 136.4859,B 24.8669,C -2.6627,E1 24.8725,E2 -52.6078} C_DIS
LIN {X -45.3646,Y 37.231,Z 72,A 133.6472,B 24.866,C -2.6712,E1 24.8774,E2 -49.7763} C_DIS
LIN {X -42.8868,Y 40.0593,Z 72,A 129.391,B 24.8661,C -2.6702,E1 24.8854,E2 -45.4986} C_DIS
LIN {X -40.3201,Y 42.642,Z 72,A 126.2857,B 24.8645,C -2.6863,E1 24.8916,E2 -42.419} C_DIS
LIN {X -38.1231,Y 44.6168,Z 72,A 123.4138,B 24.8638,C -2.693,E1 24.8976,E2 -39.5516} C_DIS
LIN {X -35.3781,Y 46.8235,Z 72,A 120.0937,B 24.8629,C -2.7023,E1 24.9049,E2 -36.2416} C_DIS
LIN {X -33.232,Y 48.371,Z 72,A 117.4938,B 24.8624,C -2.7071,E1 24.9108,E2 -33.6441} C_DIS
LIN {X -31.0564,Y 49.7948,Z 72,A 114.9311,B 24.8619,C -2.7114,E1 24.9168,E2 -31.0835} C_DIS
LIN {X -28.7616,Y 51.1549,Z 72,A 112.3642,B 24.8614,C -2.7166,E1 24.923,E2 -28.5214} C_DIS
LIN {X -26.4546,Y 52.3849,Z 72,A 109.6792,B 24.8612,C -2.7184,E1 24.9297,E2 -25.8332} C_DIS
LIN {X -24.5665,Y 53.2963,Z 72,A 107.7048,B 24.8608,C -2.7228,E1 24.9346,E2 -23.8644} C_DIS
LIN {X -22.4209,Y 54.2341,Z 72,A 104.5533,B 24.8621,C -2.7101,E1 24.9429,E2 -20.6754} C_DIS
LIN {X -18.5907,Y 55.6636,Z 72,A 101.2624,B 24.8602,C -2.728,E1 24.9514,E2 -17.4207} C_DIS
LIN {X -15.7566,Y 56.5315,Z 72,A 98.3376,B 24.86,C -2.7305,E1 24.9593,E2 -14.4971} C_DIS
LIN {X -12.9087,Y 57.2484,Z 72,A 95.2369,B 24.8602,C -2.7287,E1 24.9677,E2 -11.3879} C_DIS
LIN {X -10.3829,Y 57.76,Z 72,A 93.1365,B 24.8591,C -2.7386,E1 24.9734,E2 -9.3088} C_DIS
LIN {X -6.9663,Y 58.271,Z 72,A 90.0747,B 24.8583,C -2.7467,E1 24.9819,E2 -6.2639} C_DIS
LIN {X -5.1621,Y 58.4585,Z 72,A 87.8691,B 24.8591,C -2.7391,E1 24.988,E2 -4.0391} C_DIS
LIN {X -2.4132,Y 58.6363,Z 72,A 84.9157,B 24.8595,C -2.7349,E1 24.9963,E2 -1.0749} C_DIS
LIN {X 2.1281,Y 58.6475,Z 72,A 80.8868,B 24.8586,C -2.7436,E1 25.0075,E2 2.9328} C_DIS
LIN {X 4.5365,Y 58.5103,Z 72,A 78.3841,B 24.8589,C -2.7406,E1 25.0145,E2 5.4415} C_DIS
LIN {X 7.4055,Y 58.2169,Z 72,A 75.2366,B 24.8597,C -2.7335,E1 25.0232,E2 8.6037} C_DIS
LIN {X 10.0118,Y 57.8263,Z 72,A 72.9436,B 24.8592,C -2.7383,E1 25.0295,E2 10.883} C_DIS
LIN {X 12.9534,Y 57.2383,Z 72,A 70.373,B 24.8585,C -2.7443,E1 25.0365,E2 13.4361} C_DIS
LIN {X 15.2148,Y 56.6793,Z 72,A 67.8271,B 24.8593,C -2.7374,E1 25.0434,E2 15.9946} C_DIS
LIN {X 18.0357,Y 55.8457,Z 72,A 64.8744,B 24.8597,C -2.7336,E1 25.0513,E2 18.9511} C_DIS
LIN {X 20.9313,Y 54.8263,Z 72,A 62.0498,B 24.8596,C -2.7345,E1 25.0587,E2 21.7676} C_DIS
LIN {X 23.9786,Y 53.5633,Z 72,A 58.6095,B 24.8604,C -2.7264,E1 25.0676,E2 25.2187} C_DIS
LIN {X 27.2169,Y 51.9928,Z 72,A 55.785,B 24.8593,C -2.7368,E1 25.0746,E2 28.011} C_DIS
LIN {X 30.0535,Y 50.407,Z 72,A 51.3323,B 24.8626,C -2.705,E1 25.0855,E2 32.5259} C_DIS
LIN {X 33.1382,Y 48.4352,Z 72,A 48.6302,B 24.8612,C -2.7181,E1 25.0917,E2 35.1879} C_DIS
LIN {X 35.0966,Y 47.035,Z 72,A 46.3091,B 24.8616,C -2.7147,E1 25.0969,E2 37.5087} C_DIS
LIN {X 37.0426,Y 45.518,Z 72,A 43.7242,B 24.8624,C -2.7065,E1 25.1026,E2 40.1034} C_DIS
LIN {X 39.2072,Y 43.6672,Z 72,A 40.9413,B 24.863,C -2.7011,E1 25.1084,E2 42.8881} C_DIS
LIN {X 41.3313,Y 41.6625,Z 72,A 38.156,B 24.8634,C -2.6967,E1 25.114,E2 45.6722} C_DIS
LIN {X 43.3297,Y 39.5801,Z 72,A 35.2691,B 24.8642,C -2.6891,E1 25.1195,E2 48.5646} C_DIS
LIN {X 44.9222,Y 37.7638,Z 72,A 33.0422,B 24.8644,C -2.6867,E1 25.1236,E2 50.7871} C_DIS
LIN {X 46.6366,Y 35.6245,Z 72,A 29.6225,B 24.8668,C -2.6637,E1 25.1295,E2 54.245} C_DIS
LIN {X 49.8995,Y 30.8889,Z 72,A 25.2113,B 24.8654,C -2.6768,E1 25.1362,E2 58.6033} C_DIS
LIN {X 51.3375,Y 28.4346,Z 72,A 22.0677,B 24.867,C -2.6611,E1 25.1406,E2 61.7678} C_DIS
LIN {X 52.4709,Y 26.2847,Z 72,A 19.7494,B 24.8675,C -2.6559,E1 25.1436,E2 64.0861} C_DIS
LIN {X 53.5163,Y 24.0839,Z 72,A 17.3303,B 24.8683,C -2.6484,E1 25.1464,E2 66.5099} C_DIS
LIN {X 54.6185,Y 21.4672,Z 72,A 14.4684,B 24.8693,C -2.6384,E1 25.1495,E2 69.3796} C_DIS
LIN {X 55.5834,Y 18.8285,Z 72,A 11.9233,B 24.8696,C -2.635,E1 25.1518,E2 71.9184} C_DIS
LIN {X 56.3824,Y 16.2799,Z 72,A 8.9223,B 24.8713,C -2.6182,E1 25.1543,E2 74.9421} C_DIS
LIN {X 57.2484,Y 12.9091,Z 72,A 5.5842,B 24.8722,C -2.6093,E1 25.1564,E2 78.2819} C_DIS
LIN {X 57.9245,Y 9.4201,Z 72,A 2.2348,B 24.8729,C -2.6015,E1 25.1581,E2 81.6302} C_DIS
LIN {X 58.3486,Y 6.2849,Z 72,A -1.0296,B 24.8743,C -2.5878,E1 25.1591,E2 84.9077} C_DIS
LIN {X 58.6369,Y 2.3996,Z 72,A -4.7403,B 24.8752,C -2.578,E1 25.1597,E2 88.6195} C_DIS
LIN {X 58.6481,Y -2.1114,Z 72,A -9.6259,B 24.8777,C -2.5529,E1 25.1595,E2 93.5353} C_DIS
LIN {X 58.1065,Y -8.2258,Z 72,A -15.5445,B 24.8793,C -2.5357,E1 25.1576,E2 99.4595} C_DIS
LIN {X 56.9504,Y -14.167,Z 72,A -21.1933,B 24.8805,C -2.5233,E1 25.1542,E2 105.1049} C_DIS
LIN {X 55.9481,Y -17.715,Z 72,A -24.2668,B 24.8804,C -2.5244,E1 25.1518,E2 108.1582} C_DIS
LIN {X 55.1161,Y -20.1555,Z 72,A -26.6419,B 24.8808,C -2.52,E1 25.1496,E2 110.5303} C_DIS
LIN {X 54.1996,Y -22.5046,Z 72,A -29.393,B 24.8821,C -2.5059,E1 25.1467,E2 113.2996} C_DIS
LIN {X 52.8653,Y -25.4812,Z 72,A -32.3222,B 24.8825,C -2.5024,E1 25.1432,E2 116.2212} C_DIS
LIN {X 51.0389,Y -28.9679,Z 72,A -36.2101,B 24.8836,C -2.4902,E1 25.1381,E2 120.1175} C_DIS
LIN {X 49.5116,Y -31.5069,Z 72,A -39.3493,B 24.8849,C -2.4765,E1 25.1334,E2 123.2734} C_DIS
LIN {X 47.6813,Y -34.2132,Z 72,A -41.95,B 24.8844,C -2.4814,E1 25.1293,E2 125.8498} C_DIS
LIN {X 46.3001,Y -36.0613,Z 72,A -44.3827,B 24.8854,C -2.4712,E1 25.1252,E2 128.2949} C_DIS
LIN {X 44.6173,Y -38.1225,Z 72,A -47.075,B 24.8862,C -2.4624,E1 25.1203,E2 130.9957} C_DIS
LIN {X 42.6143,Y -40.3496,Z 72,A -49.965,B 24.8868,C -2.4559,E1 25.1149,E2 133.8883} C_DIS
LIN {X 40.5189,Y -42.4535,Z 72,A -52.8586,B 24.8874,C -2.4492,E1 25.1091,E2 136.7857} C_DIS
LIN {X 38.4752,Y -44.3138,Z 72,A -55.5458,B 24.888,C -2.4433,E1 25.1035,E2 139.4761} C_DIS
LIN {X 36.1748,Y -46.2112,Z 72,A -58.9539,B 24.8896,C -2.426,E1 25.096,E2 142.9126} C_DIS
LIN {X 32.3264,Y -48.9799,Z 72,A -63.3007,B 24.8898,C -2.423,E1 25.086,E2 147.2514} C_DIS
LIN {X 29.9325,Y -50.4785,Z 72,A -65.8095,B 24.8898,C -2.4235,E1 25.08,E2 149.7513} C_DIS
LIN {X 27.3193,Y -51.9392,Z 72,A -69.171,B 24.8911,C -2.4089,E1 25.0717,E2 153.1377} C_DIS
LIN {X 24.1156,Y -53.502,Z 72,A -72.1447,B 24.8906,C -2.4146,E1 25.0642,E2 156.0904} C_DIS
LIN {X 21.4146,Y -54.6392,Z 72,A -74.9815,B 24.8909,C -2.4111,E1 25.0569,E2 158.929} C_DIS
LIN {X 18.4856,Y -55.6986,Z 72,A -78.0521,B 24.8913,C -2.4066,E1 25.0488,E2 162.004} C_DIS
LIN {X 15.7221,Y -56.541,Z 72,A -80.9684,B 24.8918,C -2.4014,E1 25.0409,E2 164.9276} C_DIS
LIN {X 12.9067,Y -57.2489,Z 72,A -83.656,B 24.8918,C -2.4019,E1 25.0337,E2 167.6104} C_DIS
LIN {X 9.2537,Y -57.9524,Z 72,A -87.6102,B 24.8926,C -2.3923,E1 25.0227,E2 171.5831} C_DIS
LIN {X 5.9011,Y -58.3885,Z 72,A -91.5347,B 24.8939,C -2.3776,E1 25.0118,E2 175.5399} C_DIS
LIN {X 2.4881,Y -58.6331,Z 72,A -93.9737,B 24.8924,C -2.3947,E1 25.0051,E2 177.9372} C_DIS
LIN {X 0.4154,Y -58.6803,Z 72,A -95.4257,B 24.8914,C -2.406,E1 25.0011,E2 179.3623} C_DIS
Enddeposition()
LIN {X 0.4154,Y -58.6803,Z 72,A -95.4257,B 24.8914,C -2.406,E1 25.0011,E2 179.3623} C_DIS
Startdeposition()
$VEL.CP = VEL_PRINT
LIN {X 0.7036,Y -57.7035,Z 72,A -94.3303,B 24.8883,C -2.4396,E1 25.0044,E2 178.1871} C_DIS
LIN {X 3.6296,Y -57.5934,Z 72,A -91.5359,B 24.8884,C -2.4384,E1 25.0121,E2 175.3966} C_DIS
LIN {X 6.3562,Y -57.3564,Z 72,A -88.7685,B 24.8882,C -2.4409,E1 25.0198,E2 172.625} C_DIS
LIN {X 9.1418,Y -56.9795,Z 72,A -85.94,B 24.8879,C -2.4436,E1 25.0277,E2 169.7927} C_DIS
LIN {X 12.0584,Y -56.4335,Z 72,A -83.0785,B 24.8879,C -2.4443,E1 25.0355,E2 166.933} C_DIS
LIN {X 14.7942,Y -55.779,Z 72,A -80.2336,B 24.8875,C -2.4482,E1 25.0432,E2 164.0831} C_DIS
LIN {X 17.3864,Y -55.0257,Z 72,A -77.5759,B 24.8873,C -2.4508,E1 25.0503,E2 161.424} C_DIS
LIN {X 20.1046,Y -54.0921,Z 72,A -74.6811,B 24.8869,C -2.4553,E1 25.0579,E2 158.5244} C_DIS
LIN {X 22.7296,Y -53.0425,Z 72,A -71.9194,B 24.8866,C -2.4583,E1 25.0651,E2 155.762} C_DIS
LIN {X 25.324,Y -51.8539,Z 72,A -69.1157,B 24.8862,C -2.4621,E1 25.0721,E2 152.9566} C_DIS
LIN {X 27.8242,Y -50.5572,Z 72,A -66.3247,B 24.8858,C -2.4667,E1 25.079,E2 150.1627} C_DIS
LIN {X 30.2565,Y -49.1401,Z 72,A -63.5468,B 24.8854,C -2.4714,E1 25.0857,E2 147.3822} C_DIS
LIN {X 32.7016,Y -47.5479,Z 72,A -60.6538,B 24.8848,C -2.4769,E1 25.0924,E2 144.4857} C_DIS
LIN {X 34.9179,Y -45.9453,Z 72,A -57.9084,B 24.8843,C -2.4832,E1 25.0986,E2 141.7353} C_DIS
LIN {X 37.2017,Y -44.1162,Z 72,A -55.0895,B 24.8839,C -2.4876,E1 25.1047,E2 138.9167} C_DIS
LIN {X 39.277,Y -42.279,Z 72,A -52.3249,B 24.8832,C -2.4942,E1 25.1104,E2 136.1477} C_DIS
LIN {X 41.3012,Y -40.3041,Z 72,A -49.5165,B 24.8826,C -2.5009,E1 25.1159,E2 133.3353} C_DIS
LIN {X 43.2471,Y -38.2089,Z 72,A -46.6749,B 24.8819,C -2.508,E1 25.1213,E2 130.4894} C_DIS
LIN {X 45.0911,Y -36.0139,Z 72,A -43.8716,B 24.8813,C -2.5144,E1 25.1262,E2 127.6839} C_DIS
LIN {X 46.7923,Y -33.7739,Z 72,A -41.1145,B 24.8807,C -2.5211,E1 25.1308,E2 124.9244} C_DIS
LIN {X 48.3802,Y -31.4577,Z 72,A -38.3067,B 24.8799,C -2.5292,E1 25.1352,E2 122.1113} C_DIS
LIN {X 49.9108,Y -28.9672,Z 72,A -35.4452,B 24.8792,C -2.5364,E1 25.1393,E2 119.2473} C_DIS
LIN {X 51.2612,Y -26.5046,Z 72,A -32.6957,B 24.8785,C -2.5436,E1 25.1429,E2 116.4953} C_DIS
LIN {X 52.4415,Y -24.0831,Z 72,A -29.992,B 24.8777,C -2.5522,E1 25.1461,E2 113.7859} C_DIS
LIN {X 53.5816,Y -21.428,Z 72,A -27.1069,B 24.8769,C -2.5612,E1 25.1492,E2 110.8955} C_DIS
LIN {X 54.5664,Y -18.7783,Z 72,A -24.3745,B 24.8762,C -2.568,E1 25.1518,E2 108.1623} C_DIS
LIN {X 55.4207,Y -16.0831,Z 72,A -21.5865,B 24.8754,C -2.5762,E1 25.154,E2 105.3707} C_DIS
LIN {X 56.1443,Y -13.3396,Z 72,A -18.7606,B 24.8745,C -2.5852,E1 25.1559,E2 102.5399} C_DIS
LIN {X 56.7254,Y -10.602,Z 72,A -16.01,B 24.8737,C -2.5932,E1 25.1574,E2 99.7864} C_DIS
LIN {X 57.1822,Y -7.7704,Z 72,A -13.2014,B 24.873,C -2.6013,E1 25.1586,E2 96.9752} C_DIS
LIN {X 57.4997,Y -4.8986,Z 72,A -10.3074,B 24.872,C -2.611,E1 25.1594,E2 94.0755} C_DIS
LIN {X 57.6766,Y -1.8848,Z 72,A -7.3775,B 24.8712,C -2.6189,E1 25.1597,E2 91.1443} C_DIS
LIN {X 57.704,Y 0.6793,Z 72,A -4.7978,B 24.8704,C -2.6277,E1 25.1597,E2 88.5591} C_DIS
LIN {X 57.5974,Y 3.5699,Z 72,A -2.0546,B 24.8698,C -2.6337,E1 25.1593,E2 85.818} C_DIS
LIN {X 57.3537,Y 6.3797,Z 72,A 0.8048,B 24.8687,C -2.6438,E1 25.1586,E2 82.9516} C_DIS
LIN {X 56.9683,Y 9.2104,Z 72,A 3.5375,B 24.8681,C -2.6502,E1 25.1574,E2 80.22} C_DIS
LIN {X 56.4957,Y 11.7638,Z 72,A 5.9896,B 24.8676,C -2.6551,E1 25.1561,E2 77.7705} C_DIS
LIN {X 55.9795,Y 14.0157,Z 72,A 8.4448,B 24.8666,C -2.6658,E1 25.1545,E2 75.3043} C_DIS
LIN {X 55.222,Y 16.7536,Z 72,A 11.2847,B 24.8657,C -2.6747,E1 25.1523,E2 72.4597} C_DIS
LIN {X 54.3352,Y 19.4372,Z 72,A 14.0303,B 24.865,C -2.6814,E1 25.1498,E2 69.7135} C_DIS
LIN {X 53.3187,Y 22.0739,Z 72,A 16.8263,B 24.8642,C -2.6892,E1 25.1469,E2 66.9146} C_DIS
LIN {X 52.1183,Y 24.7755,Z 72,A 19.6818,B 24.8635,C -2.6955,E1 25.1436,E2 64.0596} C_DIS
LIN {X 50.8954,Y 27.2005,Z 72,A 22.4271,B 24.8627,C -2.7039,E1 25.14,E2 61.3089} C_DIS
LIN {X 49.4943,Y 29.6738,Z 72,A 25.2732,B 24.8619,C -2.7119,E1 25.136,E2 58.4587} C_DIS
LIN {X 47.9402,Y 32.1238,Z 72,A 28.0283,B 24.8614,C -2.7163,E1 25.1318,E2 55.7069} C_DIS
LIN {X 46.4099,Y 34.2974,Z 72,A 30.74,B 24.8606,C -2.7244,E1 25.1274,E2 52.9891} C_DIS
LIN {X 44.6087,Y 36.6096,Z 72,A 33.6047,B 24.86,C -2.7302,E1 25.1224,E2 50.1242} C_DIS
LIN {X 42.7524,Y 38.7618,Z 72,A 36.4579,B 24.8593,C -2.7372,E1 25.1171,E2 47.2672} C_DIS
LIN {X 40.8043,Y 40.8076,Z 72,A 39.2456,B 24.8587,C -2.7427,E1 25.1116,E2 44.4782} C_DIS
LIN {X 38.7581,Y 42.7557,Z 72,A 42.0028,B 24.8582,C -2.7473,E1 25.106,E2 41.7216} C_DIS
LIN {X 36.6189,Y 44.6011,Z 72,A 44.8082,B 24.8577,C -2.7525,E1 25.1,E2 38.9145} C_DIS
LIN {X 34.3725,Y 46.3543,Z 72,A 47.6074,B 24.8572,C -2.7568,E1 25.0938,E2 36.1152} C_DIS
LIN {X 32.0616,Y 47.9823,Z 72,A 50.4341,B 24.8567,C -2.7618,E1 25.0873,E2 33.2863} C_DIS
LIN {X 29.661,Y 49.5019,Z 72,A 53.2062,B 24.8564,C -2.765,E1 25.0807,E2 30.5156} C_DIS
LIN {X 27.1146,Y 50.941,Z 72,A 56.1153,B 24.856,C -2.769,E1 25.0735,E2 27.6054} C_DIS
LIN {X 24.6025,Y 52.2004,Z 72,A 58.8947,B 24.8557,C -2.7721,E1 25.0666,E2 24.8259} C_DIS
LIN {X 22.1395,Y 53.2916,Z 72,A 61.6061,B 24.8553,C -2.7757,E1 25.0596,E2 22.1124} C_DIS
LIN {X 19.4362,Y 54.3355,Z 72,A 64.4804,B 24.855,C -2.7783,E1 25.0521,E2 19.2381} C_DIS
LIN {X 16.7513,Y 55.2227,Z 72,A 67.2401,B 24.8549,C -2.7794,E1 25.0447,E2 16.4807} C_DIS
LIN {X 13.9175,Y 56.0041,Z 72,A 70.1092,B 24.8549,C -2.7802,E1 25.037,E2 13.6143} C_DIS
LIN {X 11.259,Y 56.5985,Z 72,A 72.8374,B 24.8546,C -2.7819,E1 25.0295,E2 10.8854} C_DIS
LIN {X 8.4567,Y 57.085,Z 72,A 75.7492,B 24.8544,C -2.7845,E1 25.0215,E2 7.9702} C_DIS
LIN {X 5.5474,Y 57.4401,Z 72,A 78.4974,B 24.8547,C -2.7817,E1 25.0139,E2 5.2306} C_DIS
LIN {X 2.8472,Y 57.6372,Z 72,A 81.2817,B 24.8544,C -2.7837,E1 25.0061,E2 2.4428} C_DIS
LIN {X -0.0753,Y 57.7079,Z 72,A 84.1483,B 24.8546,C -2.7825,E1 24.9981,E2 -0.4205} C_DIS
LIN {X -2.831,Y 57.638,Z 72,A 86.8864,B 24.8546,C -2.7817,E1 24.9905,E2 -3.1572} C_DIS
LIN {X -5.7577,Y 57.4194,Z 72,A 89.8177,B 24.8548,C -2.7806,E1 24.9823,E2 -6.0876} C_DIS
LIN {X -8.4462,Y 57.0865,Z 72,A 92.5356,B 24.8548,C -2.7795,E1 24.9748,E2 -8.8049} C_DIS
LIN {X -11.2483,Y 56.6007,Z 72,A 95.3769,B 24.8551,C -2.7777,E1 24.967,E2 -11.6448} C_DIS
LIN {X -14.0218,Y 55.978,Z 72,A 98.1846,B 24.8554,C -2.7748,E1 24.9594,E2 -14.4495} C_DIS
LIN {X -16.7434,Y 55.2251,Z 72,A 101.0369,B 24.8556,C -2.7727,E1 24.9518,E2 -17.3015} C_DIS
LIN {X -19.4243,Y 54.3398,Z 72,A 103.8076,B 24.856,C -2.7688,E1 24.9445,E2 -20.068} C_DIS
LIN {X -22.0553,Y 53.3264,Z 72,A 106.6314,B 24.8564,C -2.7654,E1 24.9371,E2 -22.8901} C_DIS
LIN {X -24.7872,Y 52.1128,Z 72,A 109.5447,B 24.8569,C -2.76,E1 24.9298,E2 -25.7975} C_DIS
Enddeposition()
END
